C07281=1125.004,205.928,-65.608,-178.986,9.407,149.569
C07282=1125.008,205.679,-65.582,-178.988,9.404,149.569
C07283=1125.013,205.431,-65.557,-178.991,9.401,149.570
C07284=1125.017,205.181,-65.532,-178.994,9.398,149.570
C07285=1125.021,204.933,-65.506,-178.997,9.395,149.570
C07286=1125.026,204.684,-65.480,-179.000,9.392,149.570
C07287=1125.030,204.435,-65.456,-179.003,9.390,149.570
C07288=1125.035,204.187,-65.431,-179.006,9.387,149.570
C07289=1125.039,203.938,-65.405,-179.009,9.383,149.570
C07290=1125.044,203.690,-65.380,-179.012,9.380,149.570
C07291=1125.048,203.441,-65.354,-179.015,9.377,149.570
C07292=1125.053,203.192,-65.330,-179.018,9.375,149.570
C07293=1125.057,202.944,-65.305,-179.021,9.371,149.571
C07294=1125.062,202.694,-65.280,-179.024,9.368,149.571
C07295=1125.066,202.446,-65.254,-179.027,9.366,149.571
C07296=1125.070,202.197,-65.230,-179.031,9.362,149.571
C07297=1125.075,201.949,-65.204,-179.033,9.359,149.571
C07298=1125.080,201.699,-65.179,-179.037,9.356,149.571
C07299=1125.084,201.451,-65.154,-179.040,9.353,149.571
C07300=1125.088,201.202,-65.130,-179.043,9.349,149.571
C07301=1125.093,200.954,-65.104,-179.046,9.347,149.572
C07302=1125.097,200.705,-65.079,-179.050,9.343,149.572
C07303=1125.102,200.456,-65.055,-179.053,9.340,149.572
C07304=1125.106,200.208,-65.029,-179.056,9.337,149.572
C07305=1125.111,199.959,-65.005,-179.060,9.333,149.572
C07306=1125.116,199.710,-64.981,-179.063,9.331,149.572
C07307=1125.119,199.496,-64.959,-179.067,9.327,149.572
C07308=1125.124,199.282,-64.937,-179.069,9.324,149.572
C07309=1125.127,199.068,-64.916,-179.072,9.321,149.572
C07310=1125.131,198.854,-64.894,-179.075,9.318,149.573
C07311=1125.135,198.640,-64.873,-179.078,9.316,149.573
C07312=1125.139,198.426,-64.852,-179.081,9.313,149.573
C07313=1125.143,198.212,-64.831,-179.084,9.309,149.573
C07314=1125.146,197.998,-64.809,-179.087,9.306,149.573
C07315=1125.151,197.750,-64.785,-179.091,9.303,149.573
C07316=1125.155,197.501,-64.760,-179.094,9.299,149.573
C07317=1125.160,197.252,-64.735,-179.098,9.296,149.573
C07318=1125.164,197.003,-64.711,-179.101,9.292,149.573
C07319=1125.169,196.754,-64.686,-179.105,9.288,149.574
C07320=1125.173,196.506,-64.662,-179.109,9.284,149.574
C07321=1125.178,196.257,-64.637,-179.112,9.281,149.574
C07322=1125.182,196.008,-64.612,-179.114,9.278,149.574
C07323=1125.187,195.760,-64.588,-179.115,9.275,149.573
C07324=1125.191,195.511,-64.563,-179.117,9.273,149.573
C07325=1125.196,195.262,-64.539,-179.119,9.270,149.573
C07326=1125.201,195.013,-64.515,-179.121,9.268,149.573
C07327=1125.205,194.764,-64.490,-179.122,9.265,149.573
C07328=1125.210,194.516,-64.465,-179.124,9.263,149.573
C07329=1125.214,194.267,-64.441,-179.125,9.260,149.572
C07330=1125.218,194.018,-64.416,-179.127,9.258,149.572
C07331=1125.223,193.769,-64.392,-179.129,9.255,149.572
C07332=1125.228,193.521,-64.368,-179.131,9.253,149.572
C07333=1125.232,193.272,-64.343,-179.133,9.249,149.572
C07334=1125.237,193.023,-64.319,-179.135,9.247,149.572
C07335=1125.241,192.774,-64.294,-179.137,9.245,149.572
C07336=1125.246,192.526,-64.270,-179.138,9.242,149.572
C07337=1125.250,192.277,-64.245,-179.140,9.240,149.572
C07338=1125.255,192.028,-64.221,-179.142,9.236,149.572
C07339=1125.259,191.780,-64.197,-179.144,9.234,149.571
C07340=1125.264,191.531,-64.173,-179.146,9.231,149.571
C07341=1125.268,191.282,-64.148,-179.148,9.228,149.571
C07342=1125.273,191.033,-64.124,-179.150,9.226,149.571
C07343=1125.278,190.784,-64.100,-179.152,9.224,149.571
C07344=1125.282,190.535,-64.076,-179.155,9.221,149.571
C07345=1125.287,190.286,-64.051,-179.156,9.218,149.571
C07346=1125.291,190.038,-64.027,-179.159,9.215,149.571
C07347=1125.295,189.790,-64.003,-179.160,9.212,149.571
C07348=1125.300,189.540,-63.979,-179.163,9.209,149.571
C07349=1125.305,189.291,-63.954,-179.165,9.207,149.571
C07350=1125.309,189.043,-63.930,-179.167,9.204,149.571
C07351=1125.313,188.794,-63.906,-179.169,9.202,149.571
C07352=1125.319,188.546,-63.882,-179.172,9.198,149.571
C07353=1125.323,188.296,-63.858,-179.174,9.195,149.571
C07354=1125.327,188.047,-63.834,-179.176,9.193,149.570
C07355=1125.332,187.799,-63.810,-179.179,9.190,149.570
C07356=1125.337,187.550,-63.785,-179.181,9.188,149.570
C07357=1125.341,187.301,-63.762,-179.183,9.184,149.570
C07358=1125.346,187.053,-63.738,-179.186,9.181,149.570
C07359=1125.350,186.804,-63.713,-179.188,9.178,149.570
C07360=1125.355,186.554,-63.689,-179.190,9.176,149.570
C07361=1125.359,186.306,-63.665,-179.193,9.173,149.570
C07362=1125.364,186.057,-63.641,-179.196,9.170,149.570
C07363=1125.368,185.843,-63.620,-179.198,9.168,149.570
C07364=1125.372,185.629,-63.600,-179.200,9.165,149.570
C07365=1125.375,185.415,-63.580,-179.202,9.162,149.570
C07366=1125.379,185.200,-63.559,-179.204,9.160,149.570
C07367=1125.383,184.987,-63.538,-179.206,9.157,149.570
C07368=1125.387,184.772,-63.517,-179.208,9.155,149.570
C07369=1125.391,184.559,-63.497,-179.211,9.153,149.570
C07370=1125.395,184.344,-63.477,-179.213,9.149,149.570
C07371=1125.399,184.096,-63.452,-179.216,9.146,149.570
C07372=1125.404,183.847,-63.429,-179.218,9.143,149.570
C07373=1125.409,183.598,-63.405,-179.221,9.140,149.570
C07374=1125.413,183.349,-63.381,-179.224,9.137,149.570
C07375=1125.418,183.100,-63.357,-179.226,9.134,149.570
C07376=1125.423,182.851,-63.333,-179.229,9.131,149.570
C07377=1125.427,182.602,-63.309,-179.231,9.128,149.570
C07378=1125.432,182.353,-63.286,-179.235,9.125,149.570
C07379=1125.436,182.105,-63.262,-179.237,9.121,149.570
C07380=1125.441,181.856,-63.238,-179.240,9.118,149.570
C07381=1125.445,181.607,-63.215,-179.242,9.115,149.570
C07382=1125.450,181.359,-63.191,-179.246,9.112,149.570
C07383=1125.454,181.109,-63.168,-179.248,9.109,149.570
C07384=1125.459,180.861,-63.144,-179.251,9.105,149.570
C07385=1125.464,180.612,-63.120,-179.254,9.102,149.570
C07386=1125.468,180.363,-63.097,-179.257,9.099,149.570
C07387=1125.473,180.115,-63.073,-179.260,9.095,149.570
C07388=1125.477,179.866,-63.049,-179.263,9.092,149.570
C07389=1125.482,179.617,-63.026,-179.265,9.089,149.570
C07390=1125.486,179.368,-63.002,-179.269,9.085,149.570
C07391=1125.491,179.118,-62.978,-179.271,9.082,149.570
C07392=1125.495,178.869,-62.955,-179.274,9.079,149.570
C07393=1125.499,178.621,-62.932,-179.275,9.076,149.570
C07394=1125.504,178.372,-62.908,-179.278,9.073,149.570
C07395=1125.509,178.124,-62.885,-179.279,9.071,149.570
C07396=1125.514,177.875,-62.862,-179.282,9.067,149.570
C07397=1125.518,177.626,-62.838,-179.284,9.064,149.570
C07398=1125.523,177.377,-62.815,-179.286,9.062,149.569
C07399=1125.527,177.128,-62.791,-179.288,9.059,149.569
C07400=1125.532,176.879,-62.768,-179.291,9.055,149.569
C07401=1125.537,176.630,-62.744,-179.292,9.053,149.569
C07402=1125.541,176.382,-62.721,-179.295,9.050,149.569
C07403=1125.545,176.133,-62.698,-179.297,9.046,149.569
C07404=1125.550,175.884,-62.675,-179.299,9.044,149.569
C07405=1125.555,175.634,-62.651,-179.301,9.041,149.569
C07406=1125.559,175.386,-62.627,-179.304,9.037,149.569
C07407=1125.564,175.137,-62.604,-179.305,9.035,149.569
C07408=1125.568,174.888,-62.581,-179.308,9.032,149.569
C07409=1125.573,174.639,-62.558,-179.310,9.029,149.568
C07410=1125.577,174.390,-62.534,-179.312,9.026,149.568
C07411=1125.582,174.141,-62.511,-179.314,9.023,149.568
C07412=1125.586,173.893,-62.488,-179.317,9.020,149.568
C07413=1125.591,173.644,-62.465,-179.318,9.017,149.568
C07414=1125.596,173.395,-62.442,-179.321,9.014,149.568
C07415=1125.601,173.146,-62.419,-179.324,9.011,149.568
C07416=1125.605,172.897,-62.395,-179.326,9.008,149.568
C07417=1125.609,172.648,-62.372,-179.327,9.005,149.568
C07418=1125.614,172.399,-62.349,-179.330,9.002,149.568
C07419=1125.618,172.185,-62.330,-179.332,9.000,149.568
C07420=1125.622,171.971,-62.309,-179.334,8.996,149.567
C07421=1125.626,171.757,-62.289,-179.336,8.994,149.567
C07422=1125.631,171.542,-62.270,-179.338,8.991,149.567
C07423=1125.634,171.328,-62.250,-179.340,8.989,149.567
C07424=1125.638,171.114,-62.230,-179.342,8.986,149.567
C07425=1125.642,170.899,-62.210,-179.344,8.983,149.567
C07426=1125.646,170.685,-62.191,-179.346,8.981,149.567
C07427=1125.651,170.436,-62.167,-179.348,8.978,149.567
C07428=1125.655,170.188,-62.145,-179.351,8.975,149.567
C07429=1125.660,169.939,-62.122,-179.352,8.972,149.567
C07430=1125.665,169.690,-62.098,-179.355,8.969,149.567
C07431=1125.669,169.441,-62.076,-179.357,8.966,149.567
C07432=1125.674,169.192,-62.053,-179.359,8.962,149.566
C07433=1125.678,168.943,-62.029,-179.362,8.959,149.566
C07434=1125.683,168.695,-62.007,-179.364,8.956,149.566
C07435=1125.688,168.446,-61.984,-179.367,8.953,149.566
C07436=1125.692,168.196,-61.962,-179.368,8.950,149.566
C07437=1125.696,167.947,-61.938,-179.371,8.947,149.566
C07438=1125.702,167.699,-61.915,-179.373,8.944,149.566
C07439=1125.706,167.450,-61.893,-179.376,8.941,149.566
C07440=1125.711,167.201,-61.870,-179.378,8.937,149.566
C07441=1125.715,166.952,-61.847,-179.380,8.934,149.566
C07442=1125.719,166.703,-61.824,-179.383,8.931,149.566
C07443=1125.724,166.454,-61.802,-179.385,8.928,149.566
C07444=1125.729,166.205,-61.779,-179.388,8.925,149.565
C07445=1125.733,165.956,-61.757,-179.389,8.922,149.565
C07446=1125.739,165.708,-61.734,-179.392,8.919,149.565
C07447=1125.743,165.459,-61.711,-179.394,8.916,149.565
C07448=1125.748,165.209,-61.688,-179.397,8.913,149.565
C07449=1125.751,164.960,-61.665,-179.399,8.910,149.565
C07450=1125.757,164.711,-61.643,-179.402,8.906,149.565
C07451=1125.761,164.463,-61.620,-179.404,8.903,149.565
C07452=1125.766,164.214,-61.597,-179.406,8.900,149.565
C07453=1125.771,163.965,-61.575,-179.409,8.897,149.565
C07454=1125.775,163.716,-61.552,-179.411,8.893,149.564
C07455=1125.780,163.467,-61.530,-179.413,8.890,149.564
C07456=1125.784,163.218,-61.507,-179.416,8.887,149.564
C07457=1125.789,162.969,-61.485,-179.418,8.884,149.564
C07458=1125.793,162.720,-61.462,-179.420,8.880,149.564
C07459=1125.798,162.471,-61.440,-179.423,8.877,149.564
C07460=1125.803,162.223,-61.417,-179.426,8.874,149.564
C07461=1125.807,161.973,-61.395,-179.428,8.871,149.564
C07462=1125.812,161.724,-61.372,-179.430,8.868,149.564
C07463=1125.817,161.476,-61.350,-179.433,8.865,149.564
C07464=1125.822,161.226,-61.327,-179.435,8.860,149.563
C07465=1125.826,160.978,-61.305,-179.438,8.857,149.563
C07466=1125.830,160.729,-61.283,-179.440,8.854,149.563
C07467=1125.835,160.479,-61.260,-179.443,8.851,149.563
C07468=1125.840,160.231,-61.238,-179.445,8.847,149.563
C07469=1125.844,159.982,-61.216,-179.448,8.844,149.563
C07470=1125.849,159.733,-61.194,-179.450,8.841,149.563
C07471=1125.854,159.484,-61.171,-179.452,8.838,149.563
C07472=1125.858,159.235,-61.149,-179.455,8.834,149.563
C07473=1125.863,158.986,-61.127,-179.457,8.830,149.563
C07474=1125.868,158.736,-61.104,-179.460,8.827,149.562
C07475=1125.872,158.522,-61.085,-179.462,8.825,149.562
C07476=1125.876,158.308,-61.066,-179.464,8.821,149.562
C07477=1125.880,158.094,-61.047,-179.466,8.818,149.562
C07478=1125.884,157.879,-61.028,-179.468,8.816,149.562
C07479=1125.888,157.665,-61.009,-179.470,8.813,149.562
C07480=1125.892,157.450,-60.990,-179.472,8.810,149.562
C07481=1125.895,157.237,-60.971,-179.475,8.807,149.562
C07482=1125.899,157.022,-60.952,-179.477,8.804,149.562
C07483=1125.904,156.773,-60.929,-179.479,8.800,149.562
C07484=1125.909,156.524,-60.908,-179.482,8.797,149.561
C07485=1125.913,156.275,-60.886,-179.484,8.794,149.561
C07486=1125.918,156.026,-60.864,-179.487,8.790,149.561
C07487=1125.922,155.777,-60.841,-179.489,8.787,149.561
C07488=1125.928,155.528,-60.819,-179.492,8.783,149.561
C07489=1125.932,155.279,-60.797,-179.494,8.779,149.561
C07490=1125.937,155.030,-60.775,-179.497,8.776,149.561
C07491=1125.941,154.781,-60.753,-179.499,8.773,149.561
C07492=1125.946,154.532,-60.731,-179.502,8.769,149.561
C07493=1125.950,154.283,-60.709,-179.504,8.765,149.560
C07494=1125.955,154.034,-60.688,-179.507,8.762,149.560
C07495=1125.960,153.785,-60.666,-179.510,8.758,149.560
C07496=1125.964,153.537,-60.644,-179.512,8.755,149.560
C07497=1125.970,153.288,-60.622,-179.514,8.751,149.560
C07498=1125.974,153.038,-60.600,-179.517,8.747,149.560
C07499=1125.979,152.790,-60.578,-179.519,8.744,149.559
C07500=1125.983,152.540,-60.556,-179.522,8.741,149.559
C07501=1125.988,152.292,-60.534,-179.525,8.736,149.559
C07502=1125.993,152.042,-60.513,-179.527,8.733,149.559
C07503=1125.998,151.793,-60.491,-179.530,8.729,149.559
C07504=1126.003,151.544,-60.470,-179.532,8.726,149.559
C07505=1126.007,151.295,-60.447,-179.535,8.722,149.559
C07506=1126.012,151.046,-60.426,-179.537,8.718,149.558
C07507=1126.016,150.797,-60.404,-179.540,8.715,149.558
C07508=1126.021,150.548,-60.382,-179.542,8.711,149.558
C07509=1126.026,150.299,-60.361,-179.545,8.707,149.558
C07510=1126.030,150.050,-60.339,-179.548,8.703,149.558
C07511=1126.035,149.801,-60.317,-179.550,8.700,149.558
C07512=1126.040,149.553,-60.296,-179.552,8.696,149.557
C07513=1126.045,149.303,-60.274,-179.555,8.693,149.557
C07514=1126.049,149.054,-60.253,-179.558,8.688,149.557
C07515=1126.054,148.806,-60.232,-179.560,8.684,149.557
C07516=1126.058,148.556,-60.210,-179.563,8.681,149.557
C07517=1126.063,148.307,-60.189,-179.566,8.677,149.557
C07518=1126.068,148.058,-60.167,-179.568,8.673,149.556
C07519=1126.072,147.809,-60.145,-179.571,8.669,149.556
C07520=1126.077,147.560,-60.124,-179.573,8.666,149.556
C07521=1126.082,147.311,-60.102,-179.576,8.662,149.556
C07522=1126.086,147.061,-60.081,-179.578,8.657,149.556
C07523=1126.091,146.813,-60.060,-179.581,8.654,149.556
C07524=1126.096,146.564,-60.038,-179.584,8.650,149.555
C07525=1126.100,146.314,-60.017,-179.586,8.646,149.555
C07526=1126.105,146.066,-59.995,-179.588,8.642,149.555
C07527=1126.110,145.816,-59.974,-179.591,8.638,149.555
C07528=1126.115,145.568,-59.953,-179.594,8.634,149.555
C07529=1126.119,145.318,-59.932,-179.596,8.631,149.555
C07530=1126.124,145.069,-59.910,-179.599,8.626,149.554
C07531=1126.128,144.855,-59.892,-179.600,8.623,149.554
C07532=1126.132,144.640,-59.874,-179.602,8.620,149.554
C07533=1126.136,144.426,-59.855,-179.603,8.618,149.553
C07534=1126.140,144.212,-59.837,-179.604,8.615,149.553
C07535=1126.145,143.997,-59.819,-179.605,8.612,149.553
C07536=1126.148,143.783,-59.801,-179.606,8.609,149.552
C07537=1126.152,143.569,-59.782,-179.608,8.606,149.552
C07538=1126.156,143.354,-59.764,-179.609,8.603,149.552
C07539=1126.161,143.105,-59.743,-179.611,8.600,149.551
C07540=1126.166,142.855,-59.721,-179.612,8.597,149.551
C07541=1126.170,142.607,-59.701,-179.613,8.594,149.551
C07542=1126.175,142.358,-59.679,-179.615,8.590,149.550
C07543=1126.180,142.109,-59.658,-179.617,8.587,149.550
C07544=1126.185,141.860,-59.638,-179.618,8.583,149.550
C07545=1126.189,141.610,-59.616,-179.619,8.580,149.549
C07546=1126.194,141.361,-59.595,-179.621,8.577,149.549
C07547=1126.198,141.112,-59.575,-179.622,8.574,149.549
C07548=1126.203,140.864,-59.553,-179.624,8.570,149.548
C07549=1126.208,140.614,-59.532,-179.625,8.567,149.548
C07550=1126.213,140.365,-59.512,-179.627,8.564,149.548
C07551=1126.217,140.116,-59.489,-179.628,8.561,149.547
C07552=1126.222,139.867,-59.469,-179.631,8.557,149.547
C07553=1126.227,139.618,-59.448,-179.632,8.554,149.547
C07554=1126.232,139.368,-59.427,-179.634,8.550,149.546
C07555=1126.236,139.120,-59.406,-179.635,8.547,149.546
C07556=1126.241,138.871,-59.385,-179.637,8.544,149.546
C07557=1126.246,138.622,-59.365,-179.638,8.540,149.545
C07558=1126.250,138.372,-59.343,-179.640,8.537,149.545
C07559=1126.255,138.123,-59.322,-179.641,8.533,149.545
C07560=1126.260,137.874,-59.301,-179.643,8.531,149.544
C07561=1126.265,137.625,-59.280,-179.645,8.527,149.544
C07562=1126.269,137.376,-59.260,-179.646,8.524,149.544
C07563=1126.274,137.127,-59.239,-179.648,8.521,149.544
C07564=1126.279,136.878,-59.219,-179.649,8.518,149.543
C07565=1126.284,136.629,-59.197,-179.651,8.514,149.543
C07566=1126.288,136.380,-59.177,-179.652,8.511,149.542
C07567=1126.293,136.130,-59.155,-179.654,8.507,149.542
C07568=1126.297,135.881,-59.135,-179.656,8.505,149.542
C07569=1126.302,135.632,-59.114,-179.657,8.501,149.542
C07570=1126.307,135.383,-59.094,-179.659,8.497,149.541
C07571=1126.312,135.134,-59.073,-179.660,8.494,149.541
C07572=1126.316,134.885,-59.052,-179.662,8.491,149.541
C07573=1126.321,134.636,-59.031,-179.664,8.488,149.540
C07574=1126.326,134.387,-59.010,-179.665,8.484,149.540
C07575=1126.331,134.138,-58.989,-179.667,8.482,149.540
C07576=1126.335,133.889,-58.969,-179.669,8.478,149.540
C07577=1126.340,133.640,-58.948,-179.671,8.474,149.539
C07578=1126.345,133.391,-58.927,-179.672,8.471,149.539
C07579=1126.349,133.142,-58.907,-179.674,8.468,149.539
C07580=1126.354,132.893,-58.886,-179.675,8.465,149.538
C07581=1126.359,132.644,-58.866,-179.677,8.461,149.538
C07582=1126.364,132.395,-58.845,-179.679,8.458,149.538
C07583=1126.368,132.146,-58.824,-179.680,8.455,149.537
C07584=1126.373,131.896,-58.805,-179.682,8.451,149.537
C07585=1126.378,131.647,-58.784,-179.684,8.449,149.537
C07586=1126.383,131.398,-58.763,-179.685,8.445,149.536
C07587=1126.387,131.183,-58.746,-179.687,8.442,149.536
C07588=1126.391,130.969,-58.727,-179.688,8.439,149.536
C07589=1126.395,130.755,-58.710,-179.690,8.437,149.536
C07590=1126.399,130.540,-58.693,-179.691,8.434,149.536
C07591=1126.403,130.325,-58.674,-179.693,8.430,149.535
C07592=1126.407,130.110,-58.657,-179.695,8.428,149.535
C07593=1126.411,129.897,-58.639,-179.696,8.425,149.535
C07594=1126.415,129.681,-58.622,-179.697,8.422,149.534
C07595=1126.421,129.432,-58.601,-179.699,8.418,149.534
C07596=1126.425,129.183,-58.581,-179.701,8.416,149.534
C07597=1126.429,128.934,-58.561,-179.703,8.412,149.534
C07598=1126.434,128.685,-58.540,-179.704,8.409,149.533
C07599=1126.439,128.435,-58.520,-179.706,8.406,149.533
C07600=1126.444,128.187,-58.500,-179.708,8.402,149.533
C07601=1126.448,127.938,-58.479,-179.709,8.399,149.532
C07602=1126.453,127.688,-58.458,-179.711,8.395,149.532
C07603=1126.458,127.439,-58.439,-179.713,8.392,149.532
C07604=1126.463,127.191,-58.419,-179.714,8.389,149.532
C07605=1126.468,126.942,-58.398,-179.716,8.385,149.531
C07606=1126.473,126.692,-58.377,-179.718,8.382,149.531
C07607=1126.478,126.443,-58.358,-179.720,8.379,149.531
C07608=1126.482,126.194,-58.337,-179.722,8.376,149.531
C07609=1126.486,125.945,-58.317,-179.724,8.372,149.530
C07610=1126.491,125.695,-58.297,-179.725,8.368,149.530
C07611=1126.496,125.446,-58.276,-179.727,8.366,149.530
C07612=1126.501,125.197,-58.256,-179.729,8.362,149.530
C07613=1126.505,124.947,-58.236,-179.731,8.359,149.529
C07614=1126.511,124.699,-58.216,-179.732,8.355,149.529
C07615=1126.515,124.450,-58.196,-179.734,8.352,149.529
C07616=1126.520,124.201,-58.176,-179.736,8.348,149.528
C07617=1126.525,123.951,-58.155,-179.738,8.346,149.528
C07618=1126.530,123.702,-58.135,-179.740,8.342,149.528
C07619=1126.534,123.453,-58.115,-179.741,8.338,149.528
C07620=1126.538,123.204,-58.095,-179.743,8.335,149.527
C07621=1126.544,122.955,-58.075,-179.745,8.332,149.527
C07622=1126.548,122.706,-58.055,-179.747,8.329,149.527
C07623=1126.553,122.457,-58.035,-179.748,8.325,149.527
C07624=1126.557,122.208,-58.015,-179.751,8.321,149.526
C07625=1126.562,121.958,-57.995,-179.752,8.319,149.526
C07626=1126.567,121.709,-57.974,-179.754,8.315,149.526
C07627=1126.573,121.460,-57.955,-179.756,8.312,149.526
C07628=1126.577,121.211,-57.935,-179.758,8.308,149.525
C07629=1126.582,120.961,-57.915,-179.759,8.305,149.525
C07630=1126.586,120.713,-57.895,-179.761,8.302,149.525
C07631=1126.591,120.463,-57.875,-179.763,8.298,149.525
C07632=1126.596,120.215,-57.855,-179.765,8.295,149.524
C07633=1126.601,119.965,-57.835,-179.767,8.291,149.524
C07634=1126.606,119.716,-57.816,-179.768,8.288,149.524
C07635=1126.610,119.467,-57.795,-179.770,8.284,149.523
C07636=1126.615,119.218,-57.776,-179.773,8.281,149.523
C07637=1126.620,118.969,-57.756,-179.775,8.277,149.523
C07638=1126.625,118.719,-57.736,-179.776,8.274,149.523
C07639=1126.629,118.470,-57.716,-179.778,8.271,149.522
C07640=1126.634,118.221,-57.696,-179.780,8.267,149.522
C07641=1126.639,117.972,-57.677,-179.782,8.264,149.522
C07642=1126.644,117.722,-57.657,-179.784,8.260,149.522
C07643=1126.648,117.508,-57.640,-179.785,8.258,149.521
C07644=1126.652,117.293,-57.623,-179.787,8.255,149.521
C07645=1126.656,117.078,-57.606,-179.789,8.251,149.521
C07646=1126.661,116.864,-57.589,-179.790,8.249,149.521
C07647=1126.664,116.649,-57.572,-179.791,8.246,149.520
C07648=1126.668,116.435,-57.556,-179.793,8.242,149.520
C07649=1126.672,116.220,-57.538,-179.795,8.239,149.520
C07650=1126.677,116.006,-57.521,-179.796,8.237,149.520
C07651=1126.681,115.756,-57.502,-179.798,8.233,149.519
C07652=1126.686,115.507,-57.482,-179.800,8.230,149.519
C07653=1126.691,115.258,-57.463,-179.802,8.226,149.519
C07654=1126.696,115.009,-57.442,-179.804,8.223,149.519
C07655=1126.701,114.759,-57.423,-179.806,8.219,149.518
C07656=1126.705,114.511,-57.404,-179.808,8.215,149.518
C07657=1126.710,114.261,-57.384,-179.810,8.212,149.518
C07658=1126.715,114.011,-57.365,-179.812,8.208,149.518
C07659=1126.720,113.763,-57.345,-179.814,8.206,149.517
C07660=1126.724,113.514,-57.325,-179.815,8.202,149.517
C07661=1126.730,113.265,-57.306,-179.817,8.198,149.517
C07662=1126.734,113.016,-57.287,-179.819,8.195,149.517
C07663=1126.739,112.766,-57.267,-179.821,8.191,149.516
C07664=1126.744,112.517,-57.248,-179.823,8.187,149.516
C07665=1126.749,112.268,-57.228,-179.825,8.184,149.516
C07666=1126.753,112.018,-57.208,-179.827,8.180,149.516
C07667=1126.758,111.769,-57.190,-179.829,8.177,149.515
C07668=1126.763,111.520,-57.170,-179.831,8.173,149.515
C07669=1126.768,111.271,-57.151,-179.833,8.169,149.515
C07670=1126.773,111.021,-57.131,-179.835,8.166,149.514
C07671=1126.778,110.772,-57.111,-179.837,8.162,149.514
C07672=1126.782,110.523,-57.093,-179.840,8.158,149.514
C07673=1126.787,110.274,-57.073,-179.842,8.155,149.514
C07674=1126.792,110.025,-57.054,-179.844,8.150,149.514
C07675=1126.796,109.776,-57.035,-179.847,8.147,149.514
C07676=1126.802,109.527,-57.015,-179.850,8.143,149.513
C07677=1126.806,109.277,-56.996,-179.852,8.139,149.513
C07678=1126.810,109.028,-56.977,-179.854,8.135,149.513
C07679=1126.816,108.779,-56.957,-179.857,8.131,149.513
C07680=1126.821,108.529,-56.938,-179.859,8.127,149.512
C07681=1126.825,108.280,-56.920,-179.862,8.123,149.512
C07682=1126.830,108.031,-56.900,-179.864,8.120,149.512
C07683=1126.835,107.782,-56.881,-179.867,8.115,149.512
C07684=1126.839,107.533,-56.862,-179.869,8.112,149.512
C07685=1126.845,107.284,-56.842,-179.871,8.107,149.511
C07686=1126.849,107.034,-56.824,-179.873,8.104,149.511
C07687=1126.854,106.785,-56.805,-179.876,8.099,149.511
C07688=1126.859,106.535,-56.785,-179.878,8.096,149.510
C07689=1126.864,106.287,-56.766,-179.880,8.092,149.510
C07690=1126.869,106.037,-56.747,-179.882,8.088,149.510
C07691=1126.873,105.788,-56.729,-179.885,8.083,149.510
C07692=1126.878,105.539,-56.709,-179.887,8.080,149.509
C07693=1126.883,105.289,-56.691,-179.889,8.076,149.509
C07694=1126.888,105.040,-56.672,-179.891,8.072,149.509
C07695=1126.892,104.791,-56.653,-179.894,8.067,149.508
C07696=1126.898,104.542,-56.634,-179.896,8.064,149.508
C07697=1126.902,104.292,-56.615,-179.898,8.060,149.508
C07698=1126.907,104.044,-56.596,-179.901,8.056,149.508
C07699=1126.912,103.829,-56.580,-179.902,8.052,149.507
C07700=1126.916,103.614,-56.563,-179.904,8.050,149.507
C07701=1126.920,103.399,-56.547,-179.906,8.046,149.507
C07702=1126.924,103.185,-56.531,-179.908,8.043,149.507
C07703=1126.928,102.969,-56.514,-179.910,8.039,149.507
C07704=1126.932,102.755,-56.499,-179.911,8.035,149.506
C07705=1126.937,102.540,-56.482,-179.913,8.032,149.506
C07706=1126.941,102.326,-56.467,-179.915,8.029,149.506
C07707=1126.945,102.076,-56.448,-179.916,8.025,149.505
C07708=1126.951,101.827,-56.429,-179.919,8.021,149.505
C07709=1126.955,101.578,-56.410,-179.921,8.017,149.505
C07710=1126.960,101.328,-56.392,-179.923,8.013,149.504
C07711=1126.965,101.080,-56.373,-179.925,8.009,149.504
C07712=1126.969,100.830,-56.355,-179.927,8.005,149.504
C07713=1126.975,100.581,-56.335,-179.929,8.001,149.503
C07714=1126.979,100.332,-56.317,-179.931,7.997,149.503
C07715=1126.985,100.081,-56.298,-179.933,7.993,149.503
C07716=1126.989,99.833,-56.280,-179.935,7.990,149.502
C07717=1126.994,99.584,-56.262,-179.937,7.985,149.502
C07718=1126.999,99.334,-56.242,-179.939,7.981,149.502
C07719=1127.004,99.085,-56.224,-179.941,7.978,149.501
C07720=1127.009,98.836,-56.206,-179.942,7.974,149.501
C07721=1127.013,98.587,-56.187,-179.945,7.969,149.501
C07722=1127.018,98.337,-56.168,-179.947,7.966,149.500
C07723=1127.023,98.088,-56.150,-179.948,7.962,149.500
C07724=1127.028,97.839,-56.132,-179.950,7.958,149.499
C07725=1127.033,97.589,-56.113,-179.953,7.954,149.499
C07726=1127.038,97.340,-56.095,-179.954,7.950,149.499
C07727=1127.043,97.091,-56.077,-179.956,7.946,149.498
C07728=1127.047,96.842,-56.058,-179.957,7.942,149.498
C07729=1127.052,96.592,-56.039,-179.959,7.938,149.498
C07730=1127.057,96.343,-56.021,-179.962,7.934,149.497
C07731=1127.062,96.094,-56.003,-179.963,7.930,149.497
C07732=1127.067,95.845,-55.985,-179.965,7.926,149.496
C07733=1127.071,95.595,-55.966,-179.967,7.922,149.496
C07734=1127.077,95.346,-55.948,-179.968,7.918,149.496
C07735=1127.082,95.097,-55.930,-179.970,7.914,149.495
C07736=1127.087,94.847,-55.912,-179.972,7.911,149.495
C07737=1127.091,94.598,-55.893,-179.974,7.906,149.495
C07738=1127.095,94.349,-55.875,-179.976,7.902,149.494
C07739=1127.100,94.100,-55.857,-179.977,7.898,149.494
C07740=1127.106,93.850,-55.838,-179.979,7.894,149.493
C07741=1127.111,93.601,-55.820,-179.980,7.890,149.493
C07742=1127.115,93.351,-55.802,-179.982,7.887,149.492
C07743=1127.120,93.102,-55.784,-179.984,7.883,149.492
C07744=1127.125,92.853,-55.766,-179.985,7.879,149.492
C07745=1127.130,92.604,-55.748,-179.987,7.875,149.491
C07746=1127.135,92.355,-55.730,-179.988,7.871,149.491
C07747=1127.140,92.105,-55.712,-179.990,7.867,149.490
C07748=1127.144,91.856,-55.693,-179.992,7.863,149.490
C07749=1127.149,91.606,-55.675,-179.993,7.859,149.489
C07750=1127.155,91.357,-55.657,-179.995,7.855,149.489
C07751=1127.160,91.108,-55.639,-179.996,7.852,149.489
C07752=1127.164,90.859,-55.621,-179.998,7.848,149.488
C07753=1127.169,90.609,-55.603,-180.000,7.844,149.488
C07754=1127.174,90.360,-55.585,179.999,7.839,149.487
C07755=1127.178,90.145,-55.570,179.997,7.836,149.487
C07756=1127.182,89.930,-55.554,179.996,7.833,149.486
C07757=1127.186,89.715,-55.538,179.995,7.830,149.486
C07758=1127.190,89.501,-55.523,179.994,7.826,149.486
C07759=1127.194,89.286,-55.508,179.993,7.823,149.485
C07760=1127.199,89.071,-55.492,179.991,7.819,149.485
C07761=1127.203,88.856,-55.476,179.990,7.816,149.484
C07762=1127.207,88.641,-55.461,179.989,7.813,149.484
C07763=1127.212,88.392,-55.443,179.988,7.809,149.483
C07764=1127.217,88.143,-55.425,179.986,7.805,149.483
C07765=1127.222,87.893,-55.408,179.984,7.801,149.483
C07766=1127.227,87.644,-55.390,179.983,7.797,149.482
C07767=1127.232,87.395,-55.372,179.982,7.793,149.481
C07768=1127.237,87.146,-55.354,179.981,7.790,149.481
C07769=1127.242,86.896,-55.336,179.979,7.786,149.481
C07770=1127.246,86.646,-55.319,179.978,7.782,149.480
C07771=1127.251,86.397,-55.301,179.976,7.778,149.480
C07772=1127.256,86.148,-55.283,179.975,7.774,149.479
C07773=1127.261,85.899,-55.265,179.973,7.770,149.479
C07774=1127.266,85.649,-55.248,179.973,7.766,149.478
C07775=1127.271,85.400,-55.230,179.971,7.762,149.478
C07776=1127.276,85.151,-55.212,179.970,7.759,149.477
C07777=1127.281,84.901,-55.194,179.968,7.754,149.477
C07778=1127.286,84.652,-55.176,179.967,7.751,149.476
C07779=1127.290,84.403,-55.159,179.966,7.747,149.476
C07780=1127.295,84.154,-55.141,179.965,7.743,149.475
C07781=1127.300,83.904,-55.124,179.963,7.739,149.475
C07782=1127.305,83.655,-55.106,179.962,7.736,149.474
C07783=1127.310,83.405,-55.088,179.961,7.732,149.474
C07784=1127.315,83.156,-55.071,179.959,7.728,149.473
C07785=1127.319,82.907,-55.053,179.959,7.724,149.472
C07786=1127.324,82.658,-55.035,179.957,7.720,149.472
C07787=1127.330,82.408,-55.018,179.956,7.716,149.472
C07788=1127.334,82.159,-55.000,179.955,7.713,149.471
C07789=1127.340,81.909,-54.983,179.954,7.709,149.471
C07790=1127.344,81.660,-54.965,179.952,7.705,149.470
C07791=1127.349,81.411,-54.947,179.952,7.702,149.470
C07792=1127.355,81.162,-54.930,179.950,7.697,149.469
C07793=1127.360,80.913,-54.912,179.949,7.694,149.468
C07794=1127.364,80.663,-54.896,179.948,7.690,149.468
C07795=1127.369,80.414,-54.878,179.947,7.687,149.467
C07796=1127.374,80.164,-54.860,179.946,7.683,149.467
C07797=1127.379,79.915,-54.842,179.945,7.679,149.466
C07798=1127.384,79.665,-54.826,179.944,7.675,149.466
C07799=1127.388,79.416,-54.808,179.943,7.671,149.465
C07800=1127.394,79.166,-54.791,179.942,7.668,149.465
C07801=1127.399,78.917,-54.773,179.940,7.664,149.464
C07802=1127.403,78.668,-54.756,179.940,7.660,149.464
C07803=1127.408,78.419,-54.738,179.938,7.657,149.463
C07804=1127.413,78.169,-54.721,179.938,7.653,149.462
C07805=1127.418,77.921,-54.704,179.936,7.649,149.462
C07806=1127.423,77.671,-54.686,179.936,7.646,149.461
C07807=1127.428,77.422,-54.668,179.935,7.641,149.461
C07808=1127.433,77.172,-54.652,179.934,7.638,149.460
C07809=1127.438,76.922,-54.634,179.933,7.635,149.460
C07810=1127.443,76.673,-54.617,179.932,7.631,149.459
C07811=1127.447,76.458,-54.602,179.931,7.628,149.459
C07812=1127.451,76.243,-54.587,179.929,7.624,149.458
C07813=1127.455,76.028,-54.572,179.928,7.621,149.458
C07814=1127.460,75.814,-54.557,179.927,7.618,149.458
C07815=1127.464,75.599,-54.543,179.926,7.614,149.457
C07816=1127.468,75.384,-54.527,179.925,7.611,149.457
C07817=1127.473,75.169,-54.513,179.923,7.607,149.456
C07818=1127.476,74.954,-54.499,179.922,7.604,149.456
C07819=1127.481,74.704,-54.481,179.920,7.600,149.455
C07820=1127.486,74.455,-54.463,179.919,7.596,149.455
C07821=1127.492,74.206,-54.447,179.917,7.592,149.455
C07822=1127.496,73.957,-54.429,179.916,7.588,149.454
C07823=1127.501,73.707,-54.412,179.915,7.584,149.453
C07824=1127.506,73.457,-54.395,179.913,7.580,149.453
C07825=1127.511,73.208,-54.378,179.911,7.576,149.453
C07826=1127.516,72.959,-54.360,179.910,7.572,149.452
C07827=1127.521,72.710,-54.344,179.909,7.568,149.452
C07828=1127.526,72.460,-54.327,179.907,7.564,149.451
C07829=1127.530,72.211,-54.310,179.906,7.560,149.451
C07830=1127.536,71.961,-54.293,179.905,7.556,149.450
C07831=1127.540,71.713,-54.276,179.903,7.552,149.450
C07832=1127.546,71.463,-54.259,179.901,7.548,149.449
C07833=1127.550,71.213,-54.242,179.900,7.544,149.449
C07834=1127.555,70.964,-54.225,179.899,7.540,149.448
C07835=1127.560,70.714,-54.208,179.897,7.536,149.448
C07836=1127.566,70.465,-54.191,179.896,7.532,149.447
C07837=1127.570,70.216,-54.175,179.894,7.527,149.447
C07838=1127.575,69.966,-54.157,179.893,7.524,149.446
C07839=1127.580,69.718,-54.140,179.891,7.520,149.446
C07840=1127.585,69.468,-54.123,179.890,7.516,149.445
C07841=1127.590,69.218,-54.106,179.889,7.511,149.445
C07842=1127.594,68.969,-54.090,179.888,7.508,149.444
C07843=1127.600,68.720,-54.073,179.886,7.504,149.444
C07844=1127.605,68.470,-54.056,179.884,7.500,149.443
C07845=1127.610,68.221,-54.039,179.883,7.496,149.443
C07846=1127.615,67.972,-54.022,179.882,7.492,149.442
C07847=1127.619,67.722,-54.006,179.880,7.488,149.442
C07848=1127.625,67.472,-53.989,179.879,7.484,149.441
C07849=1127.629,67.223,-53.972,179.878,7.480,149.441
C07850=1127.634,66.974,-53.956,179.876,7.476,149.440
C07851=1127.639,66.724,-53.938,179.875,7.472,149.440
C07852=1127.644,66.475,-53.922,179.873,7.468,149.439
C07853=1127.649,66.226,-53.905,179.872,7.464,149.439
C07854=1127.654,65.976,-53.888,179.870,7.460,149.439
C07855=1127.659,65.727,-53.871,179.869,7.456,149.438
C07856=1127.664,65.477,-53.856,179.867,7.452,149.437
C07857=1127.669,65.228,-53.839,179.866,7.448,149.437
C07858=1127.674,64.978,-53.822,179.865,7.444,149.436
C07859=1127.679,64.729,-53.806,179.863,7.440,149.436
C07860=1127.684,64.480,-53.788,179.862,7.436,149.436
C07861=1127.689,64.231,-53.772,179.861,7.432,149.435
C07862=1127.693,63.981,-53.755,179.859,7.428,149.434
C07863=1127.698,63.731,-53.739,179.857,7.424,149.434
C07864=1127.704,63.482,-53.722,179.856,7.420,149.433
C07865=1127.709,63.233,-53.706,179.855,7.416,149.433
C07866=1127.713,62.983,-53.689,179.853,7.412,149.433
C07867=1127.718,62.769,-53.675,179.852,7.409,149.432
C07868=1127.722,62.553,-53.661,179.851,7.405,149.432
C07869=1127.726,62.338,-53.646,179.850,7.402,149.431
C07870=1127.731,62.124,-53.632,179.849,7.399,149.431
C07871=1127.735,61.908,-53.618,179.847,7.395,149.430
C07872=1127.739,61.693,-53.604,179.846,7.392,149.430
C07873=1127.744,61.478,-53.590,179.845,7.388,149.430
C07874=1127.748,61.263,-53.576,179.844,7.385,149.429
C07875=1127.752,61.014,-53.559,179.843,7.380,149.428
C07876=1127.757,60.765,-53.543,179.841,7.376,149.428
C07877=1127.763,60.514,-53.526,179.840,7.372,149.427
C07878=1127.768,60.266,-53.510,179.838,7.368,149.427
C07879=1127.772,60.016,-53.494,179.837,7.364,149.427
C07880=1127.778,59.767,-53.478,179.836,7.360,149.426
C07881=1127.782,59.517,-53.461,179.834,7.356,149.425
C07882=1127.788,59.268,-53.446,179.833,7.352,149.425
C07883=1127.792,59.018,-53.429,179.832,7.348,149.424
C07884=1127.797,58.770,-53.413,179.830,7.344,149.424
C07885=1127.803,58.519,-53.396,179.829,7.340,149.423
C07886=1127.808,58.270,-53.380,179.827,7.336,149.423
C07887=1127.813,58.020,-53.364,179.826,7.332,149.422
C07888=1127.818,57.772,-53.348,179.825,7.327,149.422
C07889=1127.822,57.522,-53.331,179.823,7.324,149.421
C07890=1127.827,57.273,-53.315,179.822,7.319,149.421
C07891=1127.832,57.023,-53.299,179.820,7.315,149.420
C07892=1127.837,56.774,-53.283,179.819,7.311,149.420
C07893=1127.842,56.524,-53.266,179.818,7.307,149.419
C07894=1127.847,56.275,-53.251,179.816,7.303,149.419
C07895=1127.852,56.025,-53.234,179.815,7.299,149.418
C07896=1127.857,55.776,-53.219,179.814,7.295,149.418
C07897=1127.862,55.526,-53.202,179.812,7.291,149.417
C07898=1127.867,55.277,-53.186,179.812,7.288,149.417
C07899=1127.871,55.028,-53.170,179.810,7.284,149.416
C07900=1127.877,54.778,-53.154,179.809,7.279,149.416
C07901=1127.882,54.529,-53.138,179.807,7.275,149.415
C07902=1127.887,54.279,-53.122,179.806,7.271,149.415
C07903=1127.892,54.030,-53.106,179.805,7.267,149.414
C07904=1127.897,53.780,-53.090,179.804,7.263,149.413
C07905=1127.902,53.531,-53.074,179.802,7.259,149.413
C07906=1127.907,53.282,-53.058,179.801,7.255,149.412
C07907=1127.912,53.032,-53.042,179.799,7.251,149.412
C07908=1127.917,52.783,-53.026,179.798,7.247,149.411
C07909=1127.922,52.533,-53.010,179.797,7.243,149.411
C07910=1127.927,52.284,-52.994,179.796,7.238,149.410
C07911=1127.932,52.034,-52.978,179.794,7.234,149.410
C07912=1127.937,51.784,-52.962,179.793,7.230,149.409
C07913=1127.942,51.536,-52.946,179.791,7.226,149.409
C07914=1127.947,51.286,-52.931,179.790,7.222,149.408
C07915=1127.952,51.036,-52.915,179.789,7.218,149.408
C07916=1127.957,50.787,-52.899,179.788,7.214,149.407
C07917=1127.962,50.537,-52.883,179.786,7.210,149.407
C07918=1127.967,50.288,-52.867,179.785,7.205,149.406
C07919=1127.972,50.039,-52.852,179.783,7.202,149.406
C07920=1127.976,49.789,-52.836,179.782,7.197,149.405
C07921=1127.982,49.540,-52.820,179.781,7.193,149.404
C07922=1127.987,49.291,-52.804,179.780,7.189,149.404
C07923=1127.991,49.075,-52.791,179.778,7.185,149.403
C07924=1127.995,48.861,-52.777,179.777,7.182,149.403
C07925=1128.000,48.645,-52.763,179.776,7.178,149.403
C07926=1128.005,48.430,-52.750,179.775,7.175,149.402
C07927=1128.008,48.215,-52.736,179.774,7.171,149.401
C07928=1128.013,48.000,-52.723,179.773,7.167,149.401
C07929=1128.017,47.784,-52.710,179.772,7.164,149.401
C07930=1128.021,47.570,-52.696,179.770,7.160,149.400
C07931=1128.027,47.320,-52.681,179.769,7.156,149.400
C07932=1128.031,47.070,-52.665,179.768,7.152,149.399
C07933=1128.037,46.821,-52.649,179.767,7.148,149.398
C07934=1128.041,46.572,-52.634,179.766,7.144,149.398
C07935=1128.046,46.322,-52.618,179.764,7.140,149.397
C07936=1128.052,46.072,-52.603,179.763,7.135,149.397
C07937=1128.057,45.823,-52.587,179.761,7.131,149.396
C07938=1128.062,45.574,-52.572,179.760,7.127,149.396
C07939=1128.066,45.324,-52.556,179.759,7.123,149.395
C07940=1128.072,45.074,-52.540,179.758,7.119,149.395
C07941=1128.076,44.825,-52.525,179.757,7.115,149.394
C07942=1128.082,44.576,-52.510,179.755,7.111,149.394
C07943=1128.087,44.326,-52.494,179.754,7.106,149.393
C07944=1128.091,44.077,-52.479,179.753,7.102,149.392
C07945=1128.097,43.827,-52.463,179.751,7.098,149.392
C07946=1128.102,43.578,-52.448,179.750,7.094,149.391
C07947=1128.107,43.329,-52.433,179.749,7.090,149.391
C07948=1128.111,43.079,-52.417,179.748,7.086,149.390
C07949=1128.117,42.829,-52.401,179.747,7.081,149.389
C07950=1128.121,42.580,-52.386,179.745,7.077,149.389
C07951=1128.127,42.331,-52.371,179.744,7.073,149.388
C07952=1128.131,42.082,-52.356,179.743,7.069,149.388
C07953=1128.136,41.831,-52.340,179.741,7.065,149.387
C07954=1128.142,41.581,-52.325,179.740,7.061,149.387
C07955=1128.147,41.332,-52.310,179.739,7.056,149.386
C07956=1128.152,41.083,-52.294,179.738,7.052,149.385
C07957=1128.157,40.834,-52.279,179.737,7.048,149.385
C07958=1128.162,40.584,-52.264,179.735,7.044,149.384
C07959=1128.167,40.335,-52.249,179.734,7.039,149.384
C07960=1128.172,40.085,-52.233,179.733,7.036,149.383
C07961=1128.177,39.835,-52.218,179.732,7.031,149.383
C07962=1128.182,39.586,-52.203,179.731,7.027,149.382
C07963=1128.187,39.337,-52.187,179.730,7.023,149.381
C07964=1128.192,39.087,-52.173,179.728,7.019,149.381
C07965=1128.198,38.838,-52.157,179.727,7.014,149.380
C07966=1128.202,38.589,-52.142,179.726,7.010,149.380
C07967=1128.208,38.339,-52.127,179.724,7.006,149.379
C07968=1128.213,38.089,-52.113,179.723,7.002,149.379
C07969=1128.217,37.839,-52.097,179.722,6.997,149.378
C07970=1128.222,37.590,-52.082,179.721,6.992,149.377
C07971=1128.228,37.340,-52.067,179.719,6.988,149.377
C07972=1128.232,37.091,-52.052,179.718,6.984,149.376
C07973=1128.238,36.842,-52.036,179.717,6.980,149.376
C07974=1128.243,36.592,-52.022,179.716,6.976,149.375
C07975=1128.247,36.343,-52.007,179.715,6.971,149.374
C07976=1128.253,36.094,-51.991,179.713,6.967,149.374
C07977=1128.258,35.844,-51.977,179.712,6.963,149.373
C07978=1128.263,35.594,-51.961,179.711,6.959,149.373
C07979=1128.268,35.379,-51.948,179.711,6.955,149.372
C07980=1128.271,35.164,-51.936,179.709,6.951,149.371
C07981=1128.276,34.949,-51.923,179.708,6.948,149.371
C07982=1128.280,34.734,-51.910,179.707,6.944,149.370
C07983=1128.284,34.518,-51.897,179.706,6.941,149.370
C07984=1128.289,34.303,-51.884,179.705,6.936,149.369
C07985=1128.294,34.088,-51.871,179.704,6.933,149.369
C07986=1128.298,33.873,-51.859,179.703,6.929,149.368
C07987=1128.303,33.623,-51.844,179.702,6.925,149.368
C07988=1128.308,33.374,-51.829,179.701,6.921,149.367
C07989=1128.313,33.125,-51.814,179.699,6.916,149.367
C07990=1128.318,32.875,-51.800,179.698,6.912,149.366
C07991=1128.323,32.625,-51.785,179.697,6.908,149.365
C07992=1128.328,32.376,-51.770,179.696,6.903,149.365
C07993=1128.333,32.126,-51.755,179.695,6.899,149.364
C07994=1128.338,31.877,-51.740,179.694,6.895,149.363
C07995=1128.343,31.628,-51.725,179.692,6.890,149.363
C07996=1128.349,31.378,-51.711,179.691,6.885,149.362
C07997=1128.354,31.128,-51.696,179.690,6.881,149.362
C07998=1128.358,30.879,-51.681,179.689,6.877,149.361
C07999=1128.363,30.629,-51.667,179.688,6.873,149.360
C08000=1128.369,30.380,-51.651,179.687,6.868,149.360
C08001=1128.374,30.130,-51.637,179.686,6.864,149.359
C08002=1128.379,29.880,-51.623,179.685,6.860,149.358
C08003=1128.383,29.631,-51.608,179.684,6.856,149.358
C08004=1128.389,29.381,-51.593,179.682,6.851,149.357
C08005=1128.394,29.131,-51.579,179.681,6.847,149.356
C08006=1128.399,28.882,-51.564,179.680,6.843,149.356
C08007=1128.404,28.633,-51.549,179.679,6.837,149.355
C08008=1128.408,28.383,-51.535,179.678,6.833,149.354
C08009=1128.414,28.134,-51.520,179.677,6.829,149.354
C08010=1128.419,27.884,-51.506,179.676,6.825,149.353
C08011=1128.424,27.635,-51.491,179.674,6.820,149.352
C08012=1128.429,27.385,-51.477,179.673,6.816,149.352
C08013=1128.434,27.136,-51.462,179.672,6.812,149.351
C08014=1128.439,26.886,-51.448,179.671,6.807,149.351
C08015=1128.445,26.636,-51.433,179.670,6.803,149.350
C08016=1128.450,26.386,-51.419,179.669,6.798,149.349
C08017=1128.455,26.137,-51.405,179.668,6.794,149.349
C08018=1128.460,25.888,-51.390,179.666,6.789,149.348
C08019=1128.465,25.639,-51.376,179.665,6.785,149.347
C08020=1128.470,25.389,-51.361,179.664,6.781,149.347
C08021=1128.475,25.139,-51.347,179.664,6.776,149.346
C08022=1128.480,24.890,-51.333,179.663,6.772,149.345
C08023=1128.486,24.640,-51.318,179.662,6.767,149.345
C08024=1128.491,24.391,-51.303,179.661,6.763,149.344
C08025=1128.495,24.141,-51.289,179.659,6.758,149.343
C08026=1128.500,23.892,-51.275,179.658,6.753,149.343
C08027=1128.505,23.642,-51.260,179.657,6.749,149.342
C08028=1128.510,23.392,-51.246,179.656,6.745,149.341
C08029=1128.516,23.143,-51.232,179.655,6.741,149.341
C08030=1128.521,22.894,-51.218,179.654,6.736,149.340
C08031=1128.526,22.644,-51.204,179.653,6.732,149.339
C08032=1128.531,22.394,-51.189,179.652,6.726,149.338
C08033=1128.536,22.144,-51.175,179.650,6.722,149.338
C08034=1128.541,21.895,-51.161,179.649,6.718,149.337
C08035=1128.546,21.680,-51.149,179.649,6.714,149.337
C08036=1128.549,21.464,-51.136,179.648,6.710,149.336
C08037=1128.554,21.249,-51.124,179.646,6.706,149.335
C08038=1128.559,21.034,-51.112,179.646,6.702,149.335
C08039=1128.563,20.819,-51.099,179.645,6.698,149.334
C08040=1128.567,20.603,-51.088,179.645,6.695,149.333
C08041=1128.571,20.388,-51.076,179.643,6.690,149.333
C08042=1128.576,20.173,-51.064,179.643,6.687,149.332
C08043=1128.581,19.923,-51.049,179.641,6.682,149.332
C08044=1128.586,19.673,-51.035,179.640,6.677,149.331
C08045=1128.592,19.424,-51.021,179.639,6.673,149.330
C08046=1128.597,19.174,-51.007,179.638,6.669,149.330
C08047=1128.602,18.925,-50.993,179.638,6.664,149.329
C08048=1128.607,18.676,-50.979,179.637,6.660,149.328
C08049=1128.612,18.426,-50.965,179.635,6.654,149.327
C08050=1128.617,18.177,-50.951,179.634,6.650,149.327
C08051=1128.622,17.927,-50.937,179.633,6.645,149.326
C08052=1128.627,17.677,-50.923,179.632,6.641,149.325
C08053=1128.632,17.428,-50.909,179.631,6.637,149.325
C08054=1128.637,17.178,-50.895,179.630,6.631,149.324
C08055=1128.643,16.929,-50.881,179.629,6.627,149.323
C08056=1128.648,16.678,-50.867,179.628,6.623,149.322
C08057=1128.652,16.429,-50.853,179.628,6.618,149.322
C08058=1128.658,16.180,-50.840,179.626,6.614,149.321
C08059=1128.663,15.930,-50.825,179.625,6.609,149.320
C08060=1128.668,15.680,-50.812,179.624,6.604,149.319
C08061=1128.674,15.431,-50.798,179.623,6.599,149.319
C08062=1128.678,15.182,-50.784,179.622,6.595,149.318
C08063=1128.683,14.933,-50.770,179.622,6.590,149.317
C08064=1128.689,14.682,-50.757,179.621,6.586,149.317
C08065=1128.694,14.433,-50.742,179.619,6.581,149.316
C08066=1128.699,14.184,-50.728,179.618,6.576,149.315
C08067=1128.704,13.934,-50.716,179.618,6.572,149.314
C08068=1128.709,13.684,-50.701,179.617,6.567,149.314
C08069=1128.714,13.435,-50.687,179.615,6.562,149.313
C08070=1128.719,13.185,-50.674,179.615,6.557,149.312
C08071=1128.724,12.936,-50.660,179.614,6.553,149.311
C08072=1128.729,12.686,-50.646,179.613,6.548,149.310
C08073=1128.735,12.436,-50.633,179.612,6.544,149.310
C08074=1128.740,12.187,-50.619,179.611,6.539,149.309
C08075=1128.745,11.937,-50.606,179.610,6.534,149.308
C08076=1128.750,11.688,-50.592,179.609,6.529,149.307
C08077=1128.755,11.438,-50.578,179.608,6.525,149.307
C08078=1128.760,11.189,-50.565,179.607,6.520,149.306
C08079=1128.765,10.939,-50.551,179.606,6.515,149.305
C08080=1128.771,10.689,-50.537,179.605,6.511,149.304
C08081=1128.775,10.440,-50.524,179.604,6.506,149.304
C08082=1128.781,10.190,-50.511,179.603,6.501,149.303
C08083=1128.786,9.941,-50.496,179.602,6.496,149.302
C08084=1128.791,9.691,-50.483,179.602,6.492,149.301
C08085=1128.796,9.442,-50.469,179.601,6.487,149.300
C08086=1128.801,9.191,-50.456,179.600,6.482,149.300
C08087=1128.806,8.943,-50.443,179.599,6.477,149.299
C08088=1128.811,8.692,-50.429,179.598,6.473,149.298
C08089=1128.817,8.443,-50.416,179.597,6.468,149.297
C08090=1128.822,8.193,-50.402,179.596,6.463,149.297
C08091=1128.826,7.979,-50.391,179.596,6.459,149.296
C08092=1128.831,7.763,-50.380,179.595,6.456,149.295
C08093=1128.836,7.547,-50.368,179.596,6.452,149.294
C08094=1128.840,7.332,-50.356,179.595,6.448,149.294
C08095=1128.844,7.117,-50.344,179.595,6.443,149.293
C08096=1128.849,6.901,-50.333,179.594,6.440,149.292
C08097=1128.853,6.685,-50.322,179.594,6.436,149.291
C08098=1128.857,6.470,-50.310,179.594,6.432,149.291
C08099=1128.863,6.221,-50.297,179.593,6.428,149.290
C08100=1128.867,5.971,-50.283,179.593,6.423,149.289
C08101=1128.873,5.722,-50.270,179.592,6.418,149.288
C08102=1128.877,5.472,-50.257,179.592,6.414,149.287
C08103=1128.883,5.223,-50.243,179.591,6.410,149.286
C08104=1128.888,4.973,-50.230,179.591,6.405,149.286
C08105=1128.893,4.723,-50.217,179.590,6.400,149.285
C08106=1128.898,4.474,-50.204,179.590,6.397,149.284
C08107=1128.903,4.224,-50.190,179.590,6.392,149.283
C08108=1128.908,3.975,-50.177,179.589,6.387,149.282
C08109=1128.914,3.724,-50.164,179.589,6.382,149.281
C08110=1128.919,3.476,-50.150,179.589,6.378,149.280
C08111=1128.924,3.226,-50.137,179.588,6.374,149.280
C08112=1128.929,2.976,-50.124,179.587,6.369,149.279
C08113=1128.935,2.726,-50.111,179.587,6.365,149.278
C08114=1128.939,2.476,-50.098,179.587,6.361,149.277
C08115=1128.945,2.227,-50.084,179.586,6.356,149.276
C08116=1128.950,1.978,-50.072,179.585,6.352,149.275
C08117=1128.955,1.728,-50.058,179.585,6.347,149.275
C08118=1128.960,1.478,-50.045,179.584,6.342,149.274
C08119=1128.965,1.228,-50.032,179.584,6.338,149.273
C08120=1128.970,0.979,-50.019,179.584,6.334,149.272
C08121=1128.976,0.730,-50.006,179.583,6.329,149.271
C08122=1128.981,0.480,-49.992,179.582,6.324,149.270
C08123=1128.986,0.230,-49.980,179.582,6.320,149.269
C08124=1128.991,-0.019,-49.967,179.582,6.316,149.269
C08125=1128.996,-0.269,-49.954,179.581,6.311,149.268
C08126=1129.001,-0.519,-49.941,179.580,6.307,149.267
C08127=1129.007,-0.768,-49.927,179.580,6.302,149.266
C08128=1129.012,-1.018,-49.914,179.579,6.297,149.265
C08129=1129.017,-1.267,-49.902,179.578,6.293,149.265
C08130=1129.023,-1.517,-49.888,179.578,6.289,149.264
C08131=1129.027,-1.767,-49.875,179.578,6.284,149.263
C08132=1129.032,-2.016,-49.863,179.577,6.280,149.262
C08133=1129.038,-2.266,-49.850,179.576,6.275,149.261
C08134=1129.043,-2.516,-49.837,179.576,6.271,149.260
C08135=1129.048,-2.765,-49.824,179.575,6.266,149.260
C08136=1129.054,-3.015,-49.811,179.575,6.261,149.259
C08137=1129.058,-3.265,-49.798,179.574,6.257,149.258
C08138=1129.063,-3.514,-49.785,179.574,6.253,149.257
C08139=1129.068,-3.763,-49.773,179.573,6.248,149.256
C08140=1129.074,-4.013,-49.759,179.572,6.244,149.256
C08141=1129.079,-4.263,-49.746,179.572,6.239,149.255
C08142=1129.084,-4.512,-49.734,179.571,6.234,149.254
C08143=1129.090,-4.762,-49.721,179.570,6.230,149.253
C08144=1129.094,-5.012,-49.708,179.570,6.225,149.252
C08145=1129.099,-5.261,-49.695,179.569,6.220,149.251
C08146=1129.104,-5.511,-49.683,179.568,6.216,149.251
C08147=1129.111,-5.827,-49.667,179.567,6.210,149.250
C08148=1129.118,-6.143,-49.650,179.567,6.204,149.249
C08149=1129.125,-6.458,-49.634,179.566,6.199,149.248
C08150=1129.131,-6.774,-49.618,179.565,6.193,149.247
C08151=1129.136,-7.023,-49.605,179.564,6.188,149.246
C08152=1129.141,-7.273,-49.593,179.564,6.185,149.245
C08153=1129.146,-7.523,-49.580,179.564,6.180,149.244
C08154=1129.152,-7.772,-49.567,179.563,6.175,149.243
C08155=1129.177,-9.038,-49.501,179.448,6.358,149.317
C08156=1129.187,-9.458,-49.479,179.444,6.356,149.318
C08157=1129.191,-9.708,-49.466,179.441,6.356,149.319
C08158=1129.197,-9.958,-49.454,179.439,6.355,149.319
C08159=1129.202,-10.207,-49.442,179.436,6.354,149.320
C08160=1129.207,-10.457,-49.429,179.434,6.353,149.320
C08161=1129.213,-10.706,-49.416,179.431,6.352,149.321
C08162=1129.218,-10.956,-49.404,179.429,6.352,149.321
C08163=1129.223,-11.206,-49.391,179.427,6.351,149.322
C08164=1129.228,-11.456,-49.379,179.424,6.350,149.322
C08165=1129.233,-11.705,-49.366,179.422,6.349,149.323
C08166=1129.238,-11.955,-49.354,179.419,6.348,149.323
C08167=1129.243,-12.204,-49.342,179.417,6.348,149.324
C08168=1129.249,-12.454,-49.329,179.415,6.347,149.325
C08169=1129.253,-12.704,-49.316,179.412,6.346,149.325
C08170=1129.258,-12.953,-49.304,179.410,6.344,149.325
C08171=1129.264,-13.203,-49.292,179.407,6.344,149.326
C08172=1129.269,-13.452,-49.279,179.405,6.343,149.327
C08173=1129.274,-13.702,-49.267,179.403,6.342,149.327
C08174=1129.279,-13.951,-49.254,179.400,6.342,149.328
C08175=1129.285,-14.201,-49.241,179.398,6.341,149.328
C08176=1129.290,-14.452,-49.229,179.395,6.340,149.329
C08177=1129.295,-14.701,-49.216,179.393,6.339,149.329
C08178=1129.301,-14.951,-49.204,179.390,6.339,149.330
C08179=1129.306,-15.200,-49.192,179.388,6.338,149.330
C08180=1129.311,-15.450,-49.179,179.386,6.337,149.331
C08181=1129.316,-15.699,-49.167,179.383,6.337,149.332
C08182=1129.321,-15.949,-49.155,179.380,6.335,149.332
C08183=1129.327,-16.199,-49.143,179.378,6.334,149.332
C08184=1129.332,-16.448,-49.130,179.376,6.333,149.333
C08185=1129.337,-16.698,-49.118,179.373,6.333,149.334
C08186=1129.342,-16.947,-49.106,179.371,6.332,149.334
C08187=1129.347,-17.197,-49.093,179.369,6.331,149.335
C08188=1129.352,-17.447,-49.082,179.366,6.331,149.335
C08189=1129.357,-17.696,-49.069,179.363,6.329,149.336
C08190=1129.362,-17.946,-49.057,179.361,6.329,149.336
C08191=1129.367,-18.195,-49.044,179.359,6.328,149.337
C08192=1129.373,-18.445,-49.033,179.356,6.327,149.337
C08193=1129.378,-18.695,-49.020,179.354,6.327,149.338
C08194=1129.383,-18.945,-49.008,179.352,6.326,149.338
C08195=1129.388,-19.194,-48.996,179.349,6.325,149.339
C08196=1129.394,-19.444,-48.984,179.347,6.324,149.339
C08197=1129.399,-19.694,-48.972,179.344,6.323,149.340
C08198=1129.404,-19.943,-48.959,179.342,6.322,149.340
C08199=1129.410,-20.193,-48.947,179.340,6.322,149.341
C08200=1129.415,-20.442,-48.935,179.337,6.321,149.342
C08201=1129.420,-20.692,-48.923,179.335,6.320,149.342
C08202=1129.425,-20.941,-48.911,179.333,6.320,149.343
C08203=1129.430,-21.191,-48.899,179.330,6.319,149.343
C08204=1129.436,-21.441,-48.887,179.328,6.318,149.344
C08205=1129.441,-21.691,-48.874,179.325,6.317,149.344
C08206=1129.446,-21.941,-48.863,179.323,6.316,149.345
C08207=1129.451,-22.190,-48.850,179.320,6.316,149.345
C08208=1129.457,-22.440,-48.838,179.318,6.315,149.346
C08209=1129.461,-22.689,-48.827,179.316,6.314,149.346
C08210=1129.467,-22.939,-48.814,179.313,6.314,149.347
C08211=1129.472,-23.189,-48.802,179.311,6.313,149.347
C08212=1129.477,-23.439,-48.790,179.309,6.312,149.348
C08213=1129.483,-23.688,-48.778,179.306,6.311,149.349
C08214=1129.488,-23.938,-48.766,179.304,6.310,149.349
C08215=1129.493,-24.187,-48.755,179.301,6.309,149.350
C08216=1129.498,-24.437,-48.743,179.299,6.309,149.350
C08217=1129.504,-24.707,-48.730,179.297,6.308,149.351
C08218=1129.509,-24.977,-48.717,179.294,6.307,149.351
C08219=1129.515,-25.248,-48.704,179.291,6.306,149.352
C08220=1129.521,-25.518,-48.691,179.289,6.305,149.352
C08221=1129.526,-25.767,-48.678,179.286,6.305,149.353
C08222=1129.531,-26.017,-48.667,179.284,6.304,149.354
C08223=1129.537,-26.267,-48.655,179.282,6.303,149.354
C08224=1129.542,-26.517,-48.643,179.280,6.303,149.355
C08225=1129.546,-26.766,-48.631,179.277,6.302,149.355
C08226=1129.552,-27.015,-48.619,179.275,6.302,149.356
C08227=1129.557,-27.265,-48.608,179.273,6.301,149.356
C08228=1129.563,-27.515,-48.596,179.270,6.299,149.357
C08229=1129.567,-27.765,-48.584,179.267,6.299,149.357
C08230=1129.572,-28.014,-48.572,179.265,6.298,149.358
C08231=1129.578,-28.264,-48.560,179.263,6.297,149.358
C08232=1129.583,-28.513,-48.549,179.261,6.296,149.359
C08233=1129.589,-28.763,-48.537,179.258,6.296,149.359
C08234=1129.594,-29.013,-48.525,179.256,6.295,149.360
C08235=1129.599,-29.263,-48.513,179.254,6.294,149.360
C08236=1129.604,-29.512,-48.501,179.251,6.294,149.361
C08237=1129.609,-29.762,-48.489,179.249,6.293,149.362
C08238=1129.615,-30.012,-48.478,179.247,6.293,149.362
C08239=1129.620,-30.261,-48.467,179.244,6.292,149.363
C08240=1129.625,-30.511,-48.455,179.242,6.291,149.363
C08241=1129.631,-30.761,-48.443,179.240,6.291,149.364
C08242=1129.636,-31.010,-48.432,179.237,6.290,149.364
C08243=1129.641,-31.260,-48.420,179.235,6.288,149.365
C08244=1129.646,-31.510,-48.408,179.232,6.288,149.365
C08245=1129.651,-31.760,-48.396,179.230,6.287,149.366
C08246=1129.657,-32.009,-48.385,179.228,6.286,149.366
C08247=1129.662,-32.258,-48.373,179.225,6.285,149.367
C08248=1129.667,-32.508,-48.361,179.223,6.285,149.367
C08249=1129.672,-32.758,-48.350,179.221,6.284,149.368
C08250=1129.677,-33.008,-48.338,179.218,6.284,149.368
C08251=1129.683,-33.257,-48.326,179.216,6.283,149.369
C08252=1129.688,-33.506,-48.315,179.213,6.282,149.370
C08253=1129.693,-33.756,-48.303,179.211,6.282,149.370
C08254=1129.698,-34.006,-48.292,179.209,6.281,149.371
C08255=1129.703,-34.256,-48.280,179.206,6.280,149.371
C08256=1129.709,-34.506,-48.268,179.204,6.280,149.372
C08257=1129.714,-34.755,-48.257,179.202,6.279,149.372
C08258=1129.720,-35.005,-48.246,179.200,6.278,149.373
C08259=1129.724,-35.255,-48.235,179.197,6.278,149.373
C08260=1129.730,-35.505,-48.223,179.195,6.277,149.374
C08261=1129.735,-35.754,-48.212,179.193,6.276,149.374
C08262=1129.741,-36.004,-48.200,179.191,6.275,149.375
C08263=1129.745,-36.253,-48.189,179.188,6.275,149.376
C08264=1129.751,-36.503,-48.177,179.186,6.274,149.376
C08265=1129.755,-36.753,-48.166,179.184,6.273,149.376
C08266=1129.761,-37.002,-48.154,179.181,6.273,149.377
C08267=1129.766,-37.252,-48.143,179.179,6.272,149.378
C08268=1129.772,-37.502,-48.131,179.177,6.271,149.378
C08269=1129.777,-37.752,-48.120,179.174,6.271,149.379
C08270=1129.783,-38.001,-48.109,179.172,6.270,149.379
C08271=1129.787,-38.251,-48.098,179.170,6.270,149.380
C08272=1129.793,-38.501,-48.086,179.167,6.269,149.380
C08273=1129.797,-38.750,-48.074,179.165,6.268,149.381
C08274=1129.803,-39.000,-48.063,179.163,6.267,149.381
C08275=1129.808,-39.249,-48.052,179.160,6.267,149.382
C08276=1129.814,-39.500,-48.040,179.158,6.266,149.382
C08277=1129.819,-39.749,-48.029,179.156,6.265,149.383
C08278=1129.825,-39.999,-48.018,179.154,6.265,149.383
C08279=1129.829,-40.248,-48.006,179.151,6.264,149.384
C08280=1129.835,-40.499,-47.995,179.149,6.263,149.384
C08281=1129.840,-40.748,-47.984,179.147,6.263,149.385
C08282=1129.845,-40.997,-47.973,179.145,6.262,149.385
C08283=1129.850,-41.247,-47.961,179.142,6.261,149.386
C08284=1129.856,-41.496,-47.950,179.140,6.261,149.387
C08285=1129.862,-41.747,-47.939,179.137,6.260,149.387
C08286=1129.866,-41.996,-47.928,179.135,6.259,149.388
C08287=1129.871,-42.245,-47.917,179.133,6.259,149.388
C08288=1129.877,-42.496,-47.906,179.130,6.258,149.389
C08289=1129.882,-42.746,-47.894,179.128,6.257,149.389
C08290=1129.888,-42.995,-47.883,179.126,6.256,149.390
C08291=1129.893,-43.244,-47.871,179.123,6.256,149.390
C08292=1129.898,-43.495,-47.861,179.121,6.255,149.391
C08293=1129.904,-43.744,-47.849,179.119,6.254,149.391
C08294=1129.908,-43.993,-47.838,179.117,6.254,149.392
C08295=1129.913,-44.244,-47.827,179.114,6.253,149.393
C08296=1129.919,-44.493,-47.816,179.112,6.253,149.393
C08297=1129.924,-44.743,-47.805,179.110,6.252,149.394
C08298=1129.929,-44.993,-47.794,179.108,6.251,149.394
C08299=1129.935,-45.242,-47.783,179.105,6.251,149.395
C08300=1129.940,-45.492,-47.771,179.103,6.250,149.395
C08301=1129.945,-45.742,-47.761,179.101,6.249,149.396
C08302=1129.951,-45.991,-47.749,179.098,6.248,149.396
C08303=1129.956,-46.241,-47.739,179.096,6.248,149.397
C08304=1129.961,-46.490,-47.728,179.093,6.247,149.397
C08305=1129.967,-46.740,-47.716,179.091,6.246,149.398
C08306=1129.972,-46.991,-47.705,179.089,6.246,149.398
C08307=1129.977,-47.239,-47.694,179.087,6.245,149.399
C08308=1129.982,-47.490,-47.684,179.084,6.244,149.399
C08309=1129.988,-47.739,-47.672,179.082,6.244,149.400
C08310=1129.993,-47.989,-47.662,179.080,6.243,149.400
C08311=1129.998,-48.239,-47.650,179.078,6.243,149.401
C08312=1130.003,-48.488,-47.640,179.076,6.243,149.402
C08313=1130.009,-48.738,-47.628,179.073,6.242,149.402
C08314=1130.014,-48.988,-47.618,179.071,6.241,149.403
C08315=1130.019,-49.237,-47.607,179.069,6.240,149.403
C08316=1130.024,-49.488,-47.596,179.067,6.239,149.403
C08317=1130.030,-49.737,-47.585,179.064,6.239,149.404
C08318=1130.035,-49.987,-47.574,179.062,6.238,149.405
C08319=1130.040,-50.236,-47.563,179.060,6.238,149.405
C08320=1130.045,-50.486,-47.553,179.058,6.237,149.406
C08321=1130.051,-50.757,-47.541,179.055,6.236,149.406
C08322=1130.057,-51.028,-47.528,179.053,6.236,149.407
C08323=1130.063,-51.299,-47.516,179.050,6.235,149.408
C08324=1130.068,-51.569,-47.506,179.048,6.235,149.408
C08325=1130.073,-51.819,-47.494,179.046,6.234,149.408
C08326=1130.079,-52.069,-47.484,179.043,6.233,149.409
C08327=1130.084,-52.318,-47.472,179.041,6.233,149.410
C08328=1130.089,-52.569,-47.462,179.039,6.232,149.410
C08329=1130.095,-52.818,-47.451,179.036,6.231,149.411
C08330=1130.099,-53.068,-47.440,179.034,6.230,149.411
C08331=1130.105,-53.317,-47.430,179.032,6.230,149.412
C08332=1130.110,-53.567,-47.418,179.029,6.229,149.412
C08333=1130.116,-53.817,-47.408,179.027,6.228,149.413
C08334=1130.121,-54.067,-47.397,179.026,6.228,149.413
C08335=1130.126,-54.316,-47.386,179.023,6.228,149.414
C08336=1130.131,-54.566,-47.376,179.021,6.227,149.414
C08337=1130.137,-54.816,-47.366,179.019,6.226,149.415
C08338=1130.142,-55.065,-47.354,179.016,6.226,149.415
C08339=1130.147,-55.315,-47.344,179.014,6.225,149.416
C08340=1130.152,-55.565,-47.333,179.012,6.224,149.416
C08341=1130.158,-55.814,-47.322,179.009,6.224,149.417
C08342=1130.163,-56.065,-47.311,179.007,6.223,149.418
C08343=1130.169,-56.314,-47.301,179.005,6.222,149.418
C08344=1130.174,-56.564,-47.290,179.003,6.222,149.419
C08345=1130.179,-56.813,-47.280,179.001,6.222,149.419
C08346=1130.184,-57.064,-47.269,178.998,6.221,149.420
C08347=1130.190,-57.313,-47.259,178.996,6.220,149.420
C08348=1130.195,-57.562,-47.248,178.994,6.220,149.421
C08349=1130.200,-57.812,-47.237,178.992,6.219,149.421
C08350=1130.206,-58.062,-47.227,178.989,6.219,149.422
C08351=1130.211,-58.312,-47.217,178.987,6.218,149.422
C08352=1130.216,-58.561,-47.206,178.985,6.217,149.423
C08353=1130.221,-58.811,-47.195,178.983,6.216,149.423
C08354=1130.227,-59.061,-47.185,178.981,6.216,149.424
C08355=1130.232,-59.311,-47.174,178.978,6.216,149.424
C08356=1130.237,-59.560,-47.163,178.976,6.215,149.425
C08357=1130.242,-59.809,-47.153,178.974,6.214,149.425
C08358=1130.247,-60.060,-47.143,178.972,6.214,149.426
C08359=1130.253,-60.309,-47.132,178.970,6.213,149.426
C08360=1130.258,-60.559,-47.122,178.967,6.212,149.427
C08361=1130.264,-60.809,-47.112,178.965,6.212,149.428
C08362=1130.268,-61.059,-47.100,178.963,6.212,149.428
C08363=1130.274,-61.308,-47.090,178.961,6.211,149.429
C08364=1130.279,-61.558,-47.080,178.959,6.210,149.429
C08365=1130.284,-61.808,-47.069,178.957,6.209,149.429
C08366=1130.290,-62.058,-47.059,178.954,6.209,149.430
C08367=1130.295,-62.308,-47.049,178.952,6.208,149.431
C08368=1130.301,-62.557,-47.038,178.950,6.207,149.431
C08369=1130.306,-62.806,-47.027,178.948,6.208,149.432
C08370=1130.311,-63.056,-47.017,178.946,6.207,149.432
C08371=1130.317,-63.306,-47.007,178.943,6.206,149.433
C08372=1130.322,-63.556,-46.996,178.941,6.206,149.433
C08373=1130.326,-63.806,-46.986,178.939,6.205,149.434
C08374=1130.332,-64.055,-46.976,178.936,6.204,149.434
C08375=1130.337,-64.305,-46.966,178.934,6.203,149.435
C08376=1130.343,-64.555,-46.955,178.932,6.204,149.435
C08377=1130.348,-64.804,-46.945,178.930,6.203,149.436
C08378=1130.353,-65.055,-46.935,178.928,6.202,149.436
C08379=1130.359,-65.304,-46.925,178.926,6.201,149.437
C08380=1130.364,-65.554,-46.914,178.923,6.201,149.437
C08381=1130.369,-65.804,-46.904,178.921,6.200,149.438
C08382=1130.375,-66.054,-46.894,178.919,6.200,149.439
C08383=1130.380,-66.303,-46.884,178.917,6.200,149.439
C08384=1130.385,-66.553,-46.873,178.915,6.199,149.440
C08385=1130.390,-66.803,-46.863,178.913,6.198,149.440
C08386=1130.396,-67.052,-46.853,178.910,6.197,149.441
C08387=1130.401,-67.302,-46.842,178.908,6.197,149.441
C08388=1130.407,-67.552,-46.832,178.906,6.197,149.442
C08389=1130.412,-67.801,-46.822,178.904,6.196,149.442
C08390=1130.417,-68.051,-46.812,178.902,6.195,149.443
C08391=1130.422,-68.301,-46.802,178.900,6.195,149.443
C08392=1130.428,-68.550,-46.792,178.897,6.194,149.444
C08393=1130.433,-68.800,-46.781,178.895,6.194,149.444
C08394=1130.438,-69.050,-46.771,178.893,6.194,149.445
C08395=1130.443,-69.299,-46.761,178.891,6.193,149.445
C08396=1130.449,-69.549,-46.751,178.889,6.192,149.446
C08397=1130.454,-69.799,-46.741,178.887,6.191,149.446
C08398=1130.460,-70.049,-46.731,178.884,6.191,149.447
C08399=1130.465,-70.299,-46.721,178.882,6.190,149.447
C08400=1130.470,-70.548,-46.711,178.880,6.190,149.448
C08401=1130.475,-70.798,-46.700,178.878,6.189,149.448
C08402=1130.481,-71.048,-46.690,178.876,6.189,149.449
C08403=1130.486,-71.297,-46.680,178.874,6.188,149.449
C08404=1130.492,-71.547,-46.670,178.871,6.187,149.450
C08405=1130.496,-71.798,-46.661,178.870,6.187,149.450
C08406=1130.502,-72.047,-46.650,178.867,6.187,149.451
C08407=1130.508,-72.297,-46.640,178.865,6.186,149.452
C08408=1130.513,-72.546,-46.630,178.863,6.185,149.452
C08409=1130.518,-72.796,-46.620,178.860,6.185,149.453
C08410=1130.523,-73.046,-46.610,178.859,6.185,149.453
C08411=1130.529,-73.296,-46.600,178.857,6.184,149.453
C08412=1130.535,-73.545,-46.590,178.854,6.183,149.454
C08413=1130.540,-73.795,-46.580,178.852,6.183,149.455
C08414=1130.545,-74.045,-46.570,178.850,6.182,149.455
C08415=1130.550,-74.294,-46.560,178.848,6.182,149.456
C08416=1130.555,-74.544,-46.551,178.846,6.181,149.456
C08417=1130.561,-74.794,-46.541,178.844,6.180,149.457
C08418=1130.566,-75.043,-46.530,178.841,6.180,149.457
C08419=1130.571,-75.294,-46.520,178.839,6.179,149.458
C08420=1130.577,-75.543,-46.511,178.837,6.179,149.458
C08421=1130.582,-75.793,-46.501,178.835,6.179,149.459
C08422=1130.588,-76.043,-46.490,178.833,6.178,149.459
C08423=1130.593,-76.292,-46.482,178.831,6.177,149.460
C08424=1130.598,-76.543,-46.471,178.829,6.177,149.460
C08425=1130.604,-76.813,-46.460,178.826,6.177,149.461
C08426=1130.610,-77.085,-46.450,178.824,6.176,149.461
C08427=1130.615,-77.357,-46.439,178.822,6.175,149.462
C08428=1130.622,-77.628,-46.428,178.819,6.175,149.463
C08429=1130.626,-77.878,-46.418,178.817,6.174,149.463
C08430=1130.632,-78.128,-46.409,178.815,6.173,149.464
C08431=1130.637,-78.378,-46.399,178.813,6.173,149.464
C08432=1130.643,-78.627,-46.389,178.811,6.173,149.465
C08433=1130.649,-78.877,-46.379,178.809,6.172,149.465
C08434=1130.653,-79.127,-46.370,178.807,6.171,149.465
C08435=1130.659,-79.376,-46.360,178.804,6.171,149.466
C08436=1130.664,-79.627,-46.350,178.802,6.171,149.467
C08437=1130.669,-79.876,-46.340,178.800,6.170,149.467
C08438=1130.675,-80.126,-46.331,178.798,6.169,149.468
C08439=1130.680,-80.376,-46.321,178.796,6.169,149.468
C08440=1130.686,-80.625,-46.311,178.794,6.169,149.469
C08441=1130.691,-80.875,-46.302,178.792,6.168,149.469
C08442=1130.696,-81.125,-46.292,178.790,6.167,149.470
C08443=1130.702,-81.375,-46.282,178.787,6.167,149.470
C08444=1130.706,-81.625,-46.272,178.786,6.167,149.471
C08445=1130.712,-81.874,-46.262,178.783,6.166,149.471
C08446=1130.717,-82.124,-46.253,178.781,6.165,149.472
C08447=1130.723,-82.374,-46.243,178.779,6.165,149.472
C08448=1130.728,-82.623,-46.234,178.777,6.165,149.473
C08449=1130.734,-82.873,-46.224,178.775,6.164,149.473
C08450=1130.739,-83.123,-46.215,178.773,6.163,149.474
C08451=1130.744,-83.372,-46.205,178.771,6.162,149.474
C08452=1130.750,-83.622,-46.196,178.769,6.163,149.475
C08453=1130.755,-83.872,-46.185,178.767,6.162,149.475
C08454=1130.760,-84.122,-46.176,178.764,6.161,149.476
C08455=1130.765,-84.372,-46.166,178.763,6.161,149.476
C08456=1130.770,-84.622,-46.157,178.761,6.161,149.477
C08457=1130.776,-84.871,-46.147,178.758,6.160,149.477
C08458=1130.781,-85.121,-46.138,178.756,6.159,149.478
C08459=1130.787,-85.371,-46.128,178.755,6.159,149.478
C08460=1130.792,-85.620,-46.119,178.752,6.158,149.479
C08461=1130.798,-85.870,-46.109,178.750,6.158,149.479
C08462=1130.803,-86.120,-46.100,178.748,6.157,149.480
C08463=1130.809,-86.370,-46.090,178.746,6.157,149.480
C08464=1130.814,-86.619,-46.081,178.744,6.156,149.481
C08465=1130.819,-86.869,-46.071,178.742,6.156,149.481
C08466=1130.824,-87.119,-46.062,178.740,6.156,149.482
C08467=1130.830,-87.369,-46.052,178.738,6.155,149.482
C08468=1130.834,-87.619,-46.042,178.736,6.154,149.483
C08469=1130.840,-87.869,-46.033,178.733,6.153,149.483
C08470=1130.846,-88.119,-46.024,178.732,6.154,149.484
C08471=1130.850,-88.368,-46.014,178.730,6.153,149.484
C08472=1130.856,-88.618,-46.005,178.727,6.152,149.485
C08473=1130.861,-88.868,-45.996,178.725,6.152,149.485
C08474=1130.866,-89.117,-45.986,178.723,6.152,149.486
C08475=1130.872,-89.367,-45.977,178.721,6.151,149.486
C08476=1130.877,-89.617,-45.967,178.719,6.150,149.487
C08477=1130.883,-89.867,-45.958,178.717,6.150,149.487
C08478=1130.888,-90.117,-45.949,178.715,6.149,149.488
C08479=1130.893,-90.366,-45.939,178.713,6.149,149.488
C08480=1130.899,-90.616,-45.930,178.711,6.149,149.489
C08481=1130.904,-90.866,-45.921,178.709,6.148,149.489
C08482=1130.910,-91.115,-45.910,178.707,6.147,149.490
C08483=1130.915,-91.365,-45.902,178.705,6.147,149.490
C08484=1130.920,-91.615,-45.893,178.702,6.147,149.491
C08485=1130.926,-91.865,-45.883,178.700,6.146,149.492
C08486=1130.931,-92.115,-45.874,178.698,6.145,149.492
C08487=1130.936,-92.364,-45.865,178.696,6.146,149.493
C08488=1130.942,-92.615,-45.855,178.694,6.145,149.493
C08489=1130.947,-92.864,-45.846,178.692,6.144,149.493
C08490=1130.952,-93.113,-45.837,178.691,6.144,149.494
C08491=1130.958,-93.363,-45.828,178.688,6.143,149.494
C08492=1130.964,-93.613,-45.819,178.686,6.143,149.495
C08493=1130.969,-93.863,-45.810,178.685,6.143,149.495
C08494=1130.974,-94.112,-45.800,178.682,6.142,149.496
C08495=1130.979,-94.362,-45.791,178.680,6.141,149.496
C08496=1130.985,-94.612,-45.782,178.679,6.141,149.497
C08497=1130.990,-94.862,-45.773,178.676,6.140,149.497
C08498=1130.995,-95.111,-45.763,178.674,6.140,149.498
C08499=1131.001,-95.361,-45.754,178.672,6.140,149.499
C08500=1131.006,-95.611,-45.745,178.670,6.139,149.499
C08501=1131.012,-95.861,-45.735,178.668,6.139,149.500
C08502=1131.017,-96.111,-45.726,178.665,6.138,149.500
C08503=1131.022,-96.361,-45.718,178.664,6.138,149.501
C08504=1131.027,-96.610,-45.708,178.662,6.137,149.501
C08505=1131.033,-96.860,-45.698,178.659,6.136,149.501
C08506=1131.039,-97.110,-45.690,178.658,6.136,149.502
C08507=1131.044,-97.359,-45.681,178.656,6.136,149.502
C08508=1131.049,-97.609,-45.672,178.653,6.135,149.503
C08509=1131.055,-97.859,-45.663,178.652,6.135,149.503
C08510=1131.060,-98.109,-45.654,178.650,6.134,149.504
C08511=1131.065,-98.359,-45.644,178.647,6.133,149.504
C08512=1131.070,-98.608,-45.635,178.646,6.133,149.505
C08513=1131.076,-98.859,-45.626,178.644,6.133,149.505
C08514=1131.081,-99.108,-45.617,178.642,6.133,149.506
C08515=1131.087,-99.358,-45.608,178.640,6.132,149.506
C08516=1131.092,-99.607,-45.599,178.638,6.131,149.507
C08517=1131.098,-99.858,-45.590,178.636,6.131,149.507
C08518=1131.103,-100.107,-45.581,178.633,6.131,149.508
C08519=1131.108,-100.357,-45.572,178.631,6.130,149.509
C08520=1131.113,-100.607,-45.563,178.630,6.130,149.509
C08521=1131.119,-100.857,-45.554,178.627,6.130,149.509
C08522=1131.124,-101.106,-45.546,178.625,6.129,149.510
C08523=1131.130,-101.356,-45.536,178.624,6.129,149.510
C08524=1131.135,-101.606,-45.527,178.621,6.128,149.511
C08525=1131.141,-101.856,-45.518,178.619,6.127,149.511
C08526=1131.146,-102.106,-45.510,178.618,6.127,149.512
C08527=1131.151,-102.356,-45.501,178.615,6.127,149.512
C08528=1131.156,-102.606,-45.492,178.613,6.126,149.513
C08529=1131.162,-102.877,-45.482,178.612,6.126,149.513
C08530=1131.169,-103.150,-45.472,178.609,6.125,149.514
C08531=1131.174,-103.422,-45.462,178.607,6.124,149.514
C08532=1131.180,-103.694,-45.452,178.605,6.124,149.515
C08533=1131.185,-103.944,-45.443,178.603,6.124,149.516
C08534=1131.190,-104.194,-45.434,178.601,6.123,149.516
C08535=1131.196,-104.444,-45.426,178.599,6.123,149.517
C08536=1131.202,-104.693,-45.418,178.597,6.123,149.517
C08537=1131.207,-104.943,-45.409,178.595,6.122,149.518
C08538=1131.212,-105.193,-45.400,178.593,6.122,149.518
C08539=1131.217,-105.443,-45.391,178.591,6.121,149.518
C08540=1131.222,-105.693,-45.382,178.589,6.121,149.519
C08541=1131.229,-105.942,-45.373,178.587,6.121,149.519
C08542=1131.234,-106.192,-45.364,178.585,6.120,149.520
C08543=1131.239,-106.442,-45.355,178.583,6.119,149.520
C08544=1131.244,-106.692,-45.346,178.581,6.119,149.521
C08545=1131.249,-106.942,-45.337,178.579,6.118,149.521
C08546=1131.255,-107.191,-45.329,178.577,6.118,149.522
C08547=1131.261,-107.441,-45.321,178.575,6.118,149.522
C08548=1131.266,-107.691,-45.312,178.573,6.117,149.523
C08549=1131.271,-107.941,-45.303,178.571,6.117,149.523
C08550=1131.277,-108.190,-45.294,178.569,6.116,149.524
C08551=1131.282,-108.440,-45.285,178.568,6.116,149.524
C08552=1131.287,-108.690,-45.276,178.565,6.116,149.525
C08553=1131.292,-108.940,-45.268,178.563,6.115,149.525
C08554=1131.298,-109.189,-45.260,178.562,6.115,149.526
C08555=1131.303,-109.439,-45.251,178.559,6.114,149.526
C08556=1131.309,-109.689,-45.242,178.558,6.114,149.527
C08557=1131.314,-109.939,-45.233,178.556,6.113,149.527
C08558=1131.320,-110.188,-45.224,178.553,6.113,149.528
C08559=1131.325,-110.438,-45.216,178.552,6.113,149.528
C08560=1131.330,-110.688,-45.207,178.550,6.112,149.529
C08561=1131.335,-110.938,-45.199,178.548,6.112,149.529
C08562=1131.341,-111.187,-45.190,178.546,6.111,149.530
C08563=1131.346,-111.437,-45.181,178.544,6.111,149.530
C08564=1131.352,-111.688,-45.173,178.542,6.111,149.531
C08565=1131.357,-111.938,-45.164,178.540,6.110,149.531
C08566=1131.363,-112.187,-45.155,178.538,6.110,149.532
C08567=1131.368,-112.437,-45.147,178.537,6.109,149.532
C08568=1131.373,-112.687,-45.138,178.534,6.108,149.532
C08569=1131.379,-112.936,-45.130,178.533,6.108,149.533
C08570=1131.384,-113.186,-45.121,178.531,6.107,149.533
C08571=1131.389,-113.436,-45.112,178.529,6.107,149.534
C08572=1131.395,-113.686,-45.104,178.527,6.107,149.534
C08573=1131.401,-113.936,-45.095,178.525,6.107,149.535
C08574=1131.406,-114.185,-45.086,178.523,6.106,149.535
C08575=1131.411,-114.436,-45.078,178.521,6.105,149.536
C08576=1131.417,-114.685,-45.070,178.519,6.105,149.536
C08577=1131.422,-114.935,-45.061,178.517,6.104,149.537
C08578=1131.427,-115.185,-45.052,178.515,6.104,149.537
C08579=1131.433,-115.434,-45.045,178.513,6.104,149.538
C08580=1131.438,-115.684,-45.036,178.512,6.104,149.538
C08581=1131.443,-115.934,-45.027,178.509,6.103,149.539
C08582=1131.449,-116.184,-45.019,178.507,6.102,149.539
C08583=1131.454,-116.434,-45.010,178.506,6.102,149.540
C08584=1131.459,-116.683,-45.001,178.503,6.102,149.540
C08585=1131.466,-116.933,-44.993,178.502,6.102,149.541
C08586=1131.471,-117.183,-44.985,178.500,6.101,149.541
C08587=1131.477,-117.433,-44.977,178.498,6.101,149.542
C08588=1131.481,-117.682,-44.968,178.496,6.100,149.542
C08589=1131.486,-117.932,-44.960,178.494,6.100,149.543
C08590=1131.492,-118.182,-44.952,178.493,6.099,149.543
C08591=1131.498,-118.432,-44.943,178.490,6.098,149.543
C08592=1131.503,-118.682,-44.935,178.489,6.098,149.544
C08593=1131.509,-118.931,-44.926,178.487,6.098,149.544
C08594=1131.514,-119.181,-44.917,178.485,6.098,149.545
C08595=1131.519,-119.431,-44.910,178.483,6.097,149.545
C08596=1131.525,-119.681,-44.901,178.481,6.097,149.546
C08597=1131.530,-119.931,-44.893,178.479,6.096,149.546
C08598=1131.536,-120.180,-44.884,178.477,6.096,149.547
C08599=1131.541,-120.431,-44.876,178.475,6.096,149.547
C08600=1131.546,-120.681,-44.867,178.473,6.095,149.548
C08601=1131.551,-120.929,-44.859,178.471,6.095,149.548
C08602=1131.557,-121.180,-44.851,178.469,6.094,149.549
C08603=1131.562,-121.430,-44.842,178.468,6.094,149.549
C08604=1131.568,-121.679,-44.834,178.465,6.094,149.550
C08605=1131.573,-121.929,-44.826,178.464,6.093,149.550
C08606=1131.579,-122.179,-44.818,178.462,6.092,149.550
C08607=1131.584,-122.429,-44.809,178.460,6.092,149.551
C08608=1131.589,-122.679,-44.801,178.458,6.092,149.551
C08609=1131.595,-122.928,-44.793,178.456,6.091,149.552
C08610=1131.600,-123.178,-44.785,178.454,6.091,149.552
C08611=1131.606,-123.428,-44.777,178.452,6.090,149.553
C08612=1131.611,-123.678,-44.768,178.451,6.090,149.553
C08613=1131.617,-123.927,-44.760,178.448,6.090,149.554
C08614=1131.622,-124.177,-44.752,178.447,6.090,149.554
C08615=1131.627,-124.428,-44.744,178.445,6.089,149.555
C08616=1131.633,-124.677,-44.736,178.444,6.089,149.555
C08617=1131.638,-124.927,-44.727,178.441,6.088,149.556
C08618=1131.643,-125.176,-44.720,178.440,6.088,149.556
C08619=1131.649,-125.427,-44.711,178.438,6.087,149.557
C08620=1131.654,-125.676,-44.703,178.436,6.087,149.557
C08621=1131.660,-125.926,-44.695,178.434,6.086,149.558
C08622=1131.665,-126.176,-44.687,178.432,6.087,149.558
C08623=1131.670,-126.426,-44.678,178.430,6.086,149.559
C08624=1131.676,-126.676,-44.670,178.428,6.086,149.559
C08625=1131.681,-126.925,-44.662,178.426,6.085,149.559
C08626=1131.686,-127.175,-44.654,178.425,6.085,149.560
C08627=1131.693,-127.425,-44.646,178.423,6.084,149.560
C08628=1131.698,-127.675,-44.637,178.421,6.084,149.561
C08629=1131.703,-127.925,-44.630,178.419,6.083,149.561
C08630=1131.708,-128.174,-44.621,178.417,6.083,149.562
C08631=1131.714,-128.424,-44.614,178.415,6.083,149.562
C08632=1131.719,-128.674,-44.606,178.413,6.082,149.563
C08633=1131.298,-128.685,-44.650,178.410,6.086,149.564
C08634=1131.293,-128.435,-44.658,178.413,6.086,149.564
C08635=1131.287,-128.186,-44.666,178.414,6.087,149.564
C08636=1131.282,-127.936,-44.674,178.416,6.087,149.563
C08637=1131.277,-127.686,-44.682,178.417,6.087,149.563
C08638=1131.271,-127.436,-44.691,178.420,6.088,149.562
C08639=1131.266,-127.186,-44.699,178.421,6.088,149.562
C08640=1131.261,-126.937,-44.707,178.423,6.089,149.561
C08641=1131.255,-126.687,-44.715,178.425,6.089,149.561
C08642=1131.249,-126.437,-44.723,178.427,6.089,149.560
C08643=1131.244,-126.187,-44.732,178.429,6.089,149.560
C08644=1131.239,-125.937,-44.739,178.431,6.091,149.559
C08645=1131.234,-125.688,-44.748,178.432,6.090,149.559
C08646=1131.228,-125.438,-44.755,178.434,6.091,149.558
C08647=1131.223,-125.188,-44.763,178.436,6.091,149.558
C08648=1131.217,-124.939,-44.772,178.438,6.092,149.557
C08649=1131.212,-124.688,-44.780,178.440,6.092,149.557
C08650=1131.207,-124.438,-44.789,178.442,6.093,149.556
C08651=1131.201,-124.189,-44.796,178.444,6.093,149.556
C08652=1131.196,-123.939,-44.805,178.446,6.093,149.555
C08653=1131.190,-123.689,-44.813,178.447,6.094,149.555
C08654=1131.185,-123.439,-44.821,178.449,6.094,149.555
C08655=1131.179,-123.190,-44.829,178.451,6.095,149.554
C08656=1131.174,-122.940,-44.838,178.453,6.095,149.554
C08657=1131.169,-122.689,-44.846,178.455,6.096,149.553
C08658=1131.163,-122.440,-44.854,178.457,6.096,149.553
C08659=1131.158,-122.190,-44.862,178.459,6.096,149.552
C08660=1131.153,-121.941,-44.870,178.460,6.096,149.552
C08661=1131.147,-121.691,-44.879,178.463,6.097,149.551
C08662=1131.142,-121.441,-44.888,178.464,6.097,149.551
C08663=1131.136,-121.191,-44.895,178.466,6.098,149.550
C08664=1131.131,-120.941,-44.904,178.468,6.098,149.550
C08665=1131.125,-120.692,-44.911,178.470,6.099,149.550
C08666=1131.120,-120.442,-44.920,178.471,6.099,149.549
C08667=1131.115,-120.191,-44.929,178.474,6.100,149.549
C08668=1131.109,-119.942,-44.937,178.476,6.100,149.548
C08669=1131.103,-119.692,-44.945,178.477,6.100,149.548
C08670=1131.098,-119.443,-44.953,178.480,6.101,149.547
C08671=1131.093,-119.193,-44.962,178.481,6.101,149.547
C08672=1131.088,-118.943,-44.970,178.483,6.102,149.546
C08673=1131.082,-118.693,-44.979,178.485,6.102,149.546
C08674=1131.077,-118.443,-44.987,178.487,6.102,149.545
C08675=1131.071,-118.193,-44.996,178.489,6.102,149.545
C08676=1131.066,-117.944,-45.003,178.491,6.103,149.544
C08677=1131.061,-117.694,-45.012,178.493,6.104,149.544
C08678=1131.056,-117.444,-45.021,178.495,6.104,149.543
C08679=1131.050,-117.194,-45.029,178.496,6.105,149.543
C08680=1131.044,-116.944,-45.038,178.498,6.105,149.542
C08681=1131.039,-116.695,-45.046,178.500,6.106,149.542
C08682=1131.033,-116.445,-45.054,178.502,6.106,149.541
C08683=1131.028,-116.195,-45.063,178.504,6.106,149.541
C08684=1131.022,-115.946,-45.072,178.506,6.107,149.540
C08685=1131.018,-115.696,-45.079,178.508,6.107,149.540
C08686=1131.012,-115.446,-45.088,178.510,6.108,149.540
C08687=1131.007,-115.197,-45.097,178.512,6.108,149.539
C08688=1131.001,-114.946,-45.105,178.514,6.109,149.539
C08689=1130.996,-114.696,-45.114,178.515,6.108,149.538
C08690=1130.990,-114.447,-45.122,178.518,6.109,149.538
C08691=1130.985,-114.197,-45.131,178.520,6.110,149.537
C08692=1130.980,-113.947,-45.139,178.521,6.110,149.537
C08693=1130.974,-113.698,-45.148,178.524,6.111,149.536
C08694=1130.968,-113.447,-45.156,178.525,6.111,149.536
C08695=1130.963,-113.197,-45.165,178.527,6.111,149.535
C08696=1130.958,-112.947,-45.174,178.529,6.111,149.535
C08697=1130.952,-112.698,-45.183,178.531,6.112,149.534
C08698=1130.947,-112.448,-45.191,178.533,6.113,149.534
C08699=1130.942,-112.198,-45.200,178.535,6.113,149.533
C08700=1130.936,-111.949,-45.208,178.537,6.113,149.533
C08701=1130.931,-111.699,-45.216,178.539,6.113,149.532
C08702=1130.926,-111.449,-45.225,178.540,6.115,149.532
C08703=1130.921,-111.199,-45.234,178.543,6.115,149.531
C08704=1130.915,-110.950,-45.242,178.544,6.115,149.531
C08705=1130.910,-110.700,-45.251,178.546,6.116,149.530
C08706=1130.904,-110.449,-45.259,178.548,6.116,149.530
C08707=1130.899,-110.200,-45.268,178.550,6.117,149.530
C08708=1130.893,-109.950,-45.277,178.552,6.117,149.529
C08709=1130.888,-109.701,-45.285,178.554,6.117,149.529
C08710=1130.883,-109.451,-45.294,178.556,6.118,149.528
C08711=1130.877,-109.202,-45.303,178.558,6.118,149.528
C08712=1130.872,-108.951,-45.311,178.560,6.119,149.527
C08713=1130.866,-108.701,-45.321,178.562,6.120,149.527
C08714=1130.861,-108.451,-45.329,178.564,6.120,149.526
C08715=1130.856,-108.201,-45.338,178.566,6.120,149.526
C08716=1130.850,-107.952,-45.347,178.568,6.120,149.525
C08717=1130.845,-107.702,-45.356,178.570,6.121,149.525
C08718=1130.839,-107.452,-45.364,178.572,6.122,149.524
C08719=1130.834,-107.202,-45.373,178.574,6.122,149.524
C08720=1130.828,-106.953,-45.381,178.576,6.122,149.523
C08721=1130.823,-106.703,-45.390,178.577,6.122,149.523
C08722=1130.818,-106.453,-45.399,178.580,6.123,149.522
C08723=1130.813,-106.203,-45.408,178.582,6.124,149.522
C08724=1130.808,-105.953,-45.417,178.583,6.124,149.521
C08725=1130.802,-105.704,-45.426,178.586,6.125,149.521
C08726=1130.797,-105.454,-45.434,178.588,6.125,149.520
C08727=1130.792,-105.205,-45.443,178.589,6.125,149.520
C08728=1130.786,-104.955,-45.452,178.592,6.126,149.519
C08729=1130.780,-104.704,-45.461,178.593,6.126,149.519
C08730=1130.774,-104.455,-45.470,178.595,6.127,149.518
C08731=1130.769,-104.205,-45.478,178.598,6.127,149.518
C08732=1130.764,-103.955,-45.487,178.599,6.127,149.517
C08733=1130.759,-103.705,-45.496,178.601,6.128,149.517
C08734=1130.753,-103.433,-45.506,178.604,6.128,149.516
C08735=1130.748,-103.161,-45.516,178.606,6.129,149.516
C08736=1130.741,-102.889,-45.525,178.608,6.129,149.515
C08737=1130.735,-102.616,-45.535,178.610,6.130,149.515
C08738=1130.730,-102.366,-45.544,178.612,6.131,149.514
C08739=1130.724,-102.116,-45.553,178.614,6.131,149.514
C08740=1130.719,-101.866,-45.562,178.616,6.131,149.513
C08741=1130.714,-101.617,-45.571,178.618,6.132,149.513
C08742=1130.709,-101.367,-45.580,178.620,6.132,149.512
C08743=1130.703,-101.118,-45.589,178.622,6.133,149.512
C08744=1130.698,-100.868,-45.598,178.624,6.134,149.511
C08745=1130.693,-100.619,-45.607,178.626,6.134,149.511
C08746=1130.687,-100.368,-45.616,178.628,6.134,149.510
C08747=1130.682,-100.119,-45.625,178.630,6.135,149.510
C08748=1130.677,-99.869,-45.634,178.632,6.135,149.509
C08749=1130.672,-99.619,-45.643,178.634,6.136,149.509
C08750=1130.665,-99.369,-45.652,178.636,6.136,149.508
C08751=1130.660,-99.119,-45.661,178.638,6.136,149.508
C08752=1130.655,-98.870,-45.670,178.641,6.137,149.507
C08753=1130.650,-98.620,-45.679,178.642,6.137,149.507
C08754=1130.644,-98.370,-45.688,178.644,6.138,149.506
C08755=1130.639,-98.120,-45.697,178.646,6.138,149.506
C08756=1130.634,-97.871,-45.707,178.648,6.138,149.505
C08757=1130.629,-97.621,-45.716,178.650,6.139,149.505
C08758=1130.623,-97.371,-45.725,178.652,6.140,149.504
C08759=1130.617,-97.121,-45.734,178.654,6.140,149.504
C08760=1130.612,-96.872,-45.743,178.656,6.140,149.503
C08761=1130.606,-96.622,-45.751,178.658,6.141,149.503
C08762=1130.601,-96.372,-45.760,178.660,6.141,149.502
C08763=1130.596,-96.122,-45.771,178.662,6.142,149.502
C08764=1130.591,-95.872,-45.779,178.664,6.143,149.501
C08765=1130.585,-95.623,-45.788,178.666,6.143,149.501
C08766=1130.579,-95.372,-45.798,178.668,6.143,149.500
C08767=1130.574,-95.123,-45.807,178.670,6.144,149.500
C08768=1130.569,-94.873,-45.816,178.672,6.144,149.499
C08769=1130.564,-94.623,-45.825,178.674,6.145,149.499
C08770=1130.558,-94.373,-45.835,178.676,6.146,149.498
C08771=1130.553,-94.123,-45.844,178.679,6.146,149.498
C08772=1130.547,-93.874,-45.852,178.681,6.146,149.497
C08773=1130.542,-93.625,-45.862,178.683,6.147,149.497
C08774=1130.537,-93.375,-45.871,178.685,6.147,149.496
C08775=1130.532,-93.125,-45.880,178.687,6.147,149.496
C08776=1130.526,-92.875,-45.890,178.689,6.148,149.495
C08777=1130.520,-92.625,-45.899,178.691,6.149,149.495
C08778=1130.516,-92.376,-45.908,178.693,6.149,149.494
C08779=1130.510,-92.126,-45.918,178.695,6.150,149.494
C08780=1130.505,-91.876,-45.927,178.697,6.150,149.493
C08781=1130.500,-91.627,-45.936,178.699,6.150,149.493
C08782=1130.494,-91.376,-45.946,178.701,6.151,149.492
C08783=1130.489,-91.127,-45.955,178.703,6.152,149.492
C08784=1130.483,-90.877,-45.963,178.705,6.152,149.491
C08785=1130.478,-90.627,-45.974,178.707,6.152,149.491
C08786=1130.473,-90.377,-45.983,178.710,6.153,149.490
C08787=1130.468,-90.127,-45.992,178.712,6.154,149.490
C08788=1130.462,-89.878,-46.002,178.713,6.154,149.489
C08789=1130.457,-89.628,-46.011,178.715,6.154,149.489
C08790=1130.451,-89.378,-46.020,178.718,6.155,149.488
C08791=1130.446,-89.129,-46.030,178.719,6.155,149.488
C08792=1130.441,-88.879,-46.039,178.721,6.156,149.487
C08793=1130.435,-88.629,-46.049,178.724,6.156,149.487
C08794=1130.430,-88.379,-46.058,178.726,6.157,149.486
C08795=1130.424,-88.129,-46.067,178.727,6.157,149.486
C08796=1130.419,-87.880,-46.077,178.730,6.158,149.485
C08797=1130.413,-87.630,-46.086,178.732,6.159,149.485
C08798=1130.408,-87.380,-46.095,178.734,6.158,149.484
C08799=1130.403,-87.131,-46.105,178.736,6.159,149.484
C08800=1130.397,-86.881,-46.114,178.738,6.160,149.483
C08801=1130.393,-86.631,-46.124,178.741,6.161,149.483
C08802=1130.387,-86.381,-46.133,178.742,6.160,149.482
C08803=1130.382,-86.131,-46.143,178.744,6.161,149.482
C08804=1130.377,-85.881,-46.153,178.747,6.162,149.481
C08805=1130.371,-85.631,-46.162,178.749,6.163,149.481
C08806=1130.366,-85.382,-46.172,178.750,6.163,149.480
C08807=1130.361,-85.132,-46.181,178.752,6.163,149.480
C08808=1130.355,-84.882,-46.191,178.755,6.164,149.479
C08809=1130.350,-84.632,-46.200,178.757,6.164,149.479
C08810=1130.345,-84.383,-46.210,178.759,6.165,149.478
C08811=1130.339,-84.133,-46.219,178.761,6.165,149.478
C08812=1130.334,-83.884,-46.229,178.763,6.166,149.477
C08813=1130.328,-83.634,-46.238,178.765,6.166,149.477
C08814=1130.323,-83.384,-46.248,178.767,6.167,149.476
C08815=1130.318,-83.134,-46.257,178.769,6.167,149.476
C08816=1130.313,-82.884,-46.268,178.772,6.168,149.475
C08817=1130.307,-82.634,-46.277,178.773,6.168,149.475
C08818=1130.302,-82.385,-46.287,178.776,6.169,149.474
C08819=1130.297,-82.135,-46.296,178.778,6.169,149.474
C08820=1130.291,-81.885,-46.306,178.780,6.170,149.473
C08821=1130.286,-81.636,-46.316,178.782,6.170,149.473
C08822=1130.280,-81.386,-46.325,178.784,6.171,149.472
C08823=1130.275,-81.137,-46.335,178.786,6.172,149.472
C08824=1130.269,-80.886,-46.344,178.788,6.172,149.471
C08825=1130.264,-80.636,-46.355,178.790,6.172,149.471
C08826=1130.259,-80.386,-46.364,178.793,6.173,149.470
C08827=1130.254,-80.137,-46.374,178.795,6.173,149.469
C08828=1130.249,-79.888,-46.384,178.797,6.174,149.469
C08829=1130.243,-79.637,-46.393,178.799,6.174,149.468
C08830=1130.238,-79.388,-46.403,178.801,6.175,149.468
C08831=1130.232,-79.139,-46.413,178.803,6.176,149.468
C08832=1130.227,-78.889,-46.422,178.805,6.176,149.467
C08833=1130.222,-78.639,-46.432,178.807,6.176,149.467
C08834=1130.216,-78.388,-46.442,178.809,6.177,149.466
C08835=1130.211,-78.139,-46.452,178.812,6.177,149.465
C08836=1130.206,-77.890,-46.462,178.814,6.178,149.465
C08837=1130.200,-77.639,-46.471,178.816,6.179,149.464
C08838=1130.195,-77.368,-46.482,178.818,6.179,149.464
C08839=1130.189,-77.096,-46.493,178.820,6.179,149.463
C08840=1130.183,-76.825,-46.504,178.823,6.180,149.463
C08841=1130.177,-76.553,-46.514,178.825,6.181,149.462
C08842=1130.172,-76.304,-46.524,178.827,6.182,149.462
C08843=1130.166,-76.054,-46.534,178.829,6.182,149.461
C08844=1130.162,-75.804,-46.543,178.832,6.183,149.461
C08845=1130.156,-75.554,-46.554,178.833,6.183,149.460
C08846=1130.150,-75.305,-46.564,178.836,6.183,149.460
C08847=1130.145,-75.055,-46.574,178.838,6.184,149.459
C08848=1130.140,-74.805,-46.583,178.840,6.185,149.459
C08849=1130.135,-74.555,-46.594,178.842,6.186,149.458
C08850=1130.129,-74.306,-46.604,178.844,6.186,149.458
C08851=1130.124,-74.056,-46.613,178.846,6.186,149.457
C08852=1130.118,-73.806,-46.623,178.849,6.187,149.456
C08853=1130.113,-73.557,-46.633,178.851,6.188,149.456
C08854=1130.108,-73.306,-46.644,178.853,6.188,149.455
C08855=1130.103,-73.057,-46.653,178.855,6.188,149.455
C08856=1130.097,-72.808,-46.663,178.857,6.189,149.455
C08857=1130.091,-72.557,-46.673,178.859,6.190,149.454
C08858=1130.087,-72.307,-46.683,178.862,6.190,149.453
C08859=1130.081,-72.058,-46.693,178.864,6.191,149.453
C08860=1130.076,-71.808,-46.703,178.865,6.191,149.452
C08861=1130.070,-71.559,-46.714,178.868,6.192,149.452
C08862=1130.065,-71.309,-46.724,178.870,6.192,149.451
C08863=1130.060,-71.059,-46.733,178.872,6.193,149.451
C08864=1130.054,-70.809,-46.743,178.875,6.193,149.450
C08865=1130.049,-70.560,-46.753,178.876,6.193,149.450
C08866=1130.044,-70.309,-46.764,178.878,6.194,149.449
C08867=1130.039,-70.060,-46.774,178.881,6.195,149.449
C08868=1130.033,-69.811,-46.784,178.883,6.196,149.448
C08869=1130.028,-69.561,-46.794,178.885,6.196,149.448
C08870=1130.023,-69.311,-46.805,178.887,6.196,149.447
C08871=1130.017,-69.061,-46.815,178.889,6.197,149.447
C08872=1130.012,-68.811,-46.824,178.892,6.198,149.446
C08873=1130.007,-68.561,-46.834,178.894,6.198,149.446
C08874=1130.001,-68.312,-46.845,178.896,6.199,149.445
C08875=1129.996,-68.062,-46.855,178.898,6.200,149.445
C08876=1129.990,-67.813,-46.865,178.900,6.200,149.444
C08877=1129.985,-67.562,-46.876,178.902,6.200,149.444
C08878=1129.980,-67.313,-46.885,178.905,6.201,149.443
C08879=1129.975,-67.064,-46.895,178.907,6.202,149.443
C08880=1129.970,-66.813,-46.906,178.909,6.202,149.442
C08881=1129.964,-66.564,-46.916,178.911,6.203,149.442
C08882=1129.959,-66.314,-46.926,178.913,6.203,149.441
C08883=1129.954,-66.064,-46.937,178.915,6.204,149.440
C08884=1129.948,-65.814,-46.947,178.918,6.204,149.440
C08885=1129.943,-65.565,-46.957,178.920,6.205,149.439
C08886=1129.938,-65.315,-46.967,178.922,6.206,149.439
C08887=1129.933,-65.065,-46.978,178.924,6.207,149.438
C08888=1129.927,-64.816,-46.988,178.927,6.207,149.438
C08889=1129.922,-64.566,-46.998,178.928,6.207,149.437
C08890=1129.916,-64.316,-47.009,178.931,6.208,149.437
C08891=1129.911,-64.067,-47.019,178.933,6.209,149.436
C08892=1129.906,-63.816,-47.029,178.935,6.209,149.436
C08893=1129.900,-63.567,-47.040,178.937,6.210,149.435
C08894=1129.895,-63.317,-47.051,178.940,6.210,149.435
C08895=1129.890,-63.068,-47.061,178.941,6.210,149.434
C08896=1129.885,-62.818,-47.071,178.944,6.211,149.434
C08897=1129.880,-62.568,-47.081,178.946,6.212,149.433
C08898=1129.874,-62.319,-47.091,178.948,6.213,149.433
C08899=1129.869,-62.069,-47.102,178.951,6.213,149.432
C08900=1129.864,-61.819,-47.112,178.953,6.214,149.432
C08901=1129.858,-61.569,-47.122,178.955,6.215,149.431
C08902=1129.853,-61.319,-47.133,178.957,6.215,149.431
C08903=1129.848,-61.070,-47.144,178.959,6.215,149.430
C08904=1129.842,-60.821,-47.154,178.962,6.216,149.429
C08905=1129.837,-60.570,-47.165,178.964,6.216,149.429
C08906=1129.832,-60.321,-47.175,178.966,6.217,149.428
C08907=1129.827,-60.071,-47.185,178.968,6.218,149.428
C08908=1129.821,-59.821,-47.196,178.970,6.219,149.427
C08909=1129.816,-59.571,-47.207,178.973,6.219,149.427
C08910=1129.811,-59.322,-47.217,178.975,6.220,149.426
C08911=1129.805,-59.072,-47.227,178.977,6.220,149.426
C08912=1129.800,-58.822,-47.238,178.979,6.221,149.425
C08913=1129.795,-58.572,-47.248,178.981,6.221,149.425
C08914=1129.790,-58.323,-47.259,178.983,6.222,149.424
C08915=1129.784,-58.073,-47.270,178.986,6.222,149.424
C08916=1129.779,-57.823,-47.280,178.988,6.223,149.423
C08917=1129.774,-57.574,-47.290,178.990,6.224,149.423
C08918=1129.769,-57.324,-47.302,178.993,6.225,149.422
C08919=1129.764,-57.074,-47.312,178.995,6.226,149.422
C08920=1129.758,-56.825,-47.322,178.997,6.225,149.421
C08921=1129.753,-56.575,-47.333,178.999,6.226,149.421
C08922=1129.748,-56.326,-47.344,179.001,6.227,149.420
C08923=1129.742,-56.075,-47.355,179.003,6.227,149.420
C08924=1129.736,-55.826,-47.365,179.006,6.228,149.419
C08925=1129.732,-55.576,-47.376,179.008,6.229,149.418
C08926=1129.726,-55.326,-47.387,179.010,6.229,149.418
C08927=1129.721,-55.076,-47.397,179.013,6.230,149.417
C08928=1129.716,-54.827,-47.408,179.015,6.231,149.417
C08929=1129.711,-54.577,-47.419,179.018,6.231,149.416
C08930=1129.705,-54.327,-47.429,179.019,6.231,149.416
C08931=1129.700,-54.078,-47.440,179.021,6.232,149.415
C08932=1129.695,-53.828,-47.450,179.023,6.233,149.415
C08933=1129.689,-53.578,-47.461,179.026,6.234,149.414
C08934=1129.684,-53.329,-47.472,179.028,6.234,149.414
C08935=1129.679,-53.079,-47.483,179.031,6.235,149.413
C08936=1129.673,-52.830,-47.494,179.033,6.235,149.413
C08937=1129.669,-52.579,-47.504,179.035,6.236,149.412
C08938=1129.663,-52.330,-47.515,179.037,6.237,149.412
C08939=1129.658,-52.080,-47.526,179.040,6.237,149.411
C08940=1129.652,-51.830,-47.537,179.042,6.238,149.411
C08941=1129.647,-51.581,-47.548,179.044,6.239,149.410
C08942=1129.641,-51.309,-47.560,179.046,6.240,149.410
C08943=1129.636,-51.039,-47.571,179.049,6.240,149.409
C08944=1129.630,-50.768,-47.583,179.051,6.241,149.408
C08945=1129.625,-50.497,-47.595,179.054,6.241,149.408
C08946=1129.619,-50.248,-47.606,179.056,6.242,149.407
C08947=1129.614,-49.998,-47.617,179.058,6.243,149.407
C08948=1129.609,-49.748,-47.627,179.060,6.243,149.406
C08949=1129.603,-49.499,-47.639,179.063,6.244,149.406
C08950=1129.598,-49.249,-47.649,179.065,6.245,149.405
C08951=1129.593,-48.999,-47.660,179.068,6.245,149.405
C08952=1129.588,-48.749,-47.671,179.069,6.245,149.404
C08953=1129.582,-48.500,-47.683,179.071,6.246,149.404
C08954=1129.577,-48.250,-47.693,179.074,6.247,149.403
C08955=1129.572,-48.001,-47.704,179.076,6.247,149.402
C08956=1129.567,-47.750,-47.715,179.078,6.248,149.402
C08957=1129.561,-47.501,-47.727,179.081,6.249,149.401
C08958=1129.556,-47.251,-47.737,179.083,6.249,149.401
C08959=1129.551,-47.001,-47.748,179.085,6.250,149.400
C08960=1129.545,-46.751,-47.759,179.088,6.251,149.400
C08961=1129.540,-46.502,-47.770,179.090,6.252,149.399
C08962=1129.535,-46.252,-47.781,179.092,6.252,149.399
C08963=1129.530,-46.003,-47.792,179.095,6.253,149.398
C08964=1129.524,-45.753,-47.804,179.097,6.253,149.398
C08965=1129.519,-45.503,-47.814,179.099,6.254,149.397
C08966=1129.514,-45.254,-47.825,179.101,6.255,149.397
C08967=1129.508,-45.004,-47.837,179.104,6.255,149.396
C08968=1129.503,-44.754,-47.847,179.106,6.256,149.396
C08969=1129.498,-44.504,-47.858,179.108,6.257,149.395
C08970=1129.493,-44.255,-47.870,179.110,6.258,149.395
C08971=1129.487,-44.005,-47.880,179.113,6.258,149.394
C08972=1129.482,-43.755,-47.892,179.115,6.259,149.393
C08973=1129.477,-43.505,-47.904,179.117,6.260,149.393
C08974=1129.471,-43.256,-47.914,179.120,6.260,149.392
C08975=1129.467,-43.006,-47.925,179.122,6.261,149.392
C08976=1129.461,-42.756,-47.937,179.125,6.262,149.391
C08977=1129.456,-42.507,-47.947,179.127,6.262,149.391
C08978=1129.450,-42.257,-47.959,179.129,6.263,149.390
C08979=1129.446,-42.007,-47.970,179.132,6.263,149.390
C08980=1129.440,-41.758,-47.981,179.134,6.264,149.389
C08981=1129.435,-41.508,-47.993,179.136,6.265,149.389
C08982=1129.430,-41.258,-48.004,179.138,6.266,149.388
C08983=1129.424,-41.009,-48.015,179.140,6.267,149.388
C08984=1129.419,-40.759,-48.027,179.143,6.267,149.387
C08985=1129.414,-40.509,-48.037,179.145,6.268,149.387
C08986=1129.409,-40.259,-48.049,179.147,6.268,149.386
C08987=1129.403,-40.010,-48.060,179.149,6.268,149.386
C08988=1129.398,-39.760,-48.072,179.152,6.269,149.385
C08989=1129.393,-39.511,-48.083,179.154,6.270,149.384
C08990=1129.387,-39.261,-48.094,179.157,6.271,149.384
C08991=1129.382,-39.011,-48.105,179.159,6.272,149.383
C08992=1129.377,-38.761,-48.117,179.161,6.272,149.383
C08993=1129.372,-38.512,-48.128,179.164,6.273,149.382
C08994=1129.366,-38.262,-48.140,179.166,6.274,149.382
C08995=1129.361,-38.013,-48.151,179.168,6.275,149.381
C08996=1129.356,-37.762,-48.162,179.171,6.275,149.381
C08997=1129.350,-37.513,-48.173,179.173,6.276,149.380
C08998=1129.345,-37.263,-48.185,179.175,6.277,149.380
C08999=1129.340,-37.014,-48.197,179.177,6.277,149.379
C09000=1129.335,-36.764,-48.208,179.180,6.278,149.378
C09001=1129.330,-36.515,-48.219,179.182,6.279,149.378
C09002=1129.324,-36.265,-48.231,179.184,6.279,149.378
C09003=1129.319,-36.015,-48.243,179.186,6.280,149.377
C09004=1129.314,-35.765,-48.254,179.189,6.281,149.376
C09005=1129.309,-35.515,-48.265,179.191,6.281,149.376
C09006=1129.303,-35.266,-48.276,179.194,6.282,149.375
C09007=1129.298,-35.016,-48.288,179.196,6.283,149.375
C09008=1129.293,-34.766,-48.300,179.198,6.283,149.374
C09009=1129.288,-34.517,-48.311,179.201,6.284,149.374
C09010=1129.283,-34.267,-48.323,179.203,6.285,149.373
C09011=1129.277,-34.017,-48.334,179.205,6.286,149.373
C09012=1129.272,-33.768,-48.346,179.208,6.286,149.372
C09013=1129.267,-33.518,-48.358,179.210,6.287,149.372
C09014=1129.262,-33.268,-48.369,179.212,6.288,149.371
C09015=1129.256,-33.018,-48.381,179.215,6.288,149.370
C09016=1129.251,-32.769,-48.392,179.217,6.289,149.370
C09017=1129.246,-32.519,-48.404,179.219,6.289,149.370
C09018=1129.240,-32.270,-48.415,179.221,6.290,149.369
C09019=1129.236,-32.020,-48.427,179.224,6.291,149.368
C09020=1129.230,-31.770,-48.439,179.226,6.291,149.368
C09021=1129.225,-31.520,-48.450,179.228,6.292,149.367
C09022=1129.219,-31.271,-48.461,179.230,6.293,149.367
C09023=1129.214,-31.022,-48.474,179.233,6.293,149.366
C09024=1129.210,-30.772,-48.485,179.236,6.295,149.366
C09025=1129.204,-30.522,-48.497,179.238,6.296,149.365
C09026=1129.199,-30.272,-48.509,179.240,6.296,149.365
C09027=1129.194,-30.023,-48.520,179.243,6.297,149.364
C09028=1129.189,-29.773,-48.532,179.245,6.298,149.364
C09029=1129.183,-29.523,-48.544,179.247,6.298,149.363
C09030=1129.178,-29.274,-48.555,179.249,6.299,149.363
C09031=1129.172,-29.024,-48.567,179.252,6.300,149.362
C09032=1129.167,-28.775,-48.580,179.254,6.300,149.361
C09033=1129.163,-28.525,-48.591,179.257,6.301,149.361
C09034=1129.157,-28.275,-48.603,179.259,6.302,149.361
C09035=1129.152,-28.025,-48.615,179.261,6.302,149.360
C09036=1129.146,-27.775,-48.626,179.264,6.303,149.359
C09037=1129.142,-27.526,-48.638,179.266,6.304,149.359
C09038=1129.136,-27.277,-48.650,179.269,6.305,149.358
C09039=1129.131,-27.027,-48.662,179.271,6.306,149.358
C09040=1129.126,-26.777,-48.673,179.273,6.307,149.357
C09041=1129.120,-26.527,-48.685,179.276,6.307,149.357
C09042=1129.115,-26.277,-48.697,179.278,6.308,149.356
C09043=1129.110,-26.028,-48.710,179.280,6.309,149.356
C09044=1129.105,-25.779,-48.721,179.283,6.309,149.355
C09045=1129.100,-25.529,-48.733,179.285,6.310,149.355
C09046=1129.094,-25.258,-48.746,179.287,6.311,149.354
C09047=1129.089,-24.989,-48.758,179.290,6.312,149.353
C09048=1129.082,-24.718,-48.772,179.293,6.313,149.353
C09049=1129.077,-24.448,-48.785,179.295,6.313,149.352
C09050=1129.072,-24.199,-48.796,179.298,6.314,149.352
C09051=1129.067,-23.949,-48.808,179.300,6.314,149.351
C09052=1129.061,-23.699,-48.820,179.303,6.316,149.351
C09053=1129.056,-23.449,-48.832,179.305,6.317,149.350
C09054=1129.051,-23.200,-48.845,179.308,6.317,149.349
C09055=1129.045,-22.950,-48.857,179.310,6.318,149.349
C09056=1129.041,-22.701,-48.868,179.312,6.319,149.349
C09057=1129.036,-22.451,-48.880,179.314,6.320,149.348
C09058=1129.030,-22.201,-48.892,179.317,6.320,149.347
C09059=1129.025,-21.951,-48.904,179.319,6.321,149.347
C09060=1129.020,-21.702,-48.917,179.321,6.322,149.346
C09061=1129.014,-21.452,-48.929,179.324,6.323,149.346
C09062=1129.009,-21.203,-48.941,179.327,6.324,149.345
C09063=1129.004,-20.953,-48.953,179.329,6.324,149.345
C09064=1128.999,-20.703,-48.965,179.331,6.325,149.344
C09065=1128.994,-20.454,-48.977,179.334,6.325,149.344
C09066=1128.988,-20.204,-48.989,179.336,6.326,149.343
C09067=1128.983,-19.955,-49.002,179.338,6.327,149.343
C09068=1128.978,-19.705,-49.013,179.341,6.327,149.342
C09069=1128.973,-19.455,-49.026,179.343,6.329,149.342
C09070=1128.967,-19.206,-49.038,179.346,6.330,149.341
C09071=1128.962,-18.956,-49.050,179.348,6.331,149.341
C09072=1128.957,-18.706,-49.062,179.350,6.331,149.340
C09073=1128.951,-18.456,-49.074,179.353,6.332,149.339
C09074=1128.929,-17.334,-49.132,179.540,6.000,149.212
C09075=1128.924,-17.085,-49.144,179.541,6.004,149.212
C09076=1128.918,-16.835,-49.156,179.542,6.009,149.213
C09077=1128.914,-16.586,-49.168,179.542,6.013,149.214
C09078=1128.908,-16.336,-49.180,179.543,6.019,149.215
C09079=1128.903,-16.087,-49.193,179.544,6.023,149.216
C09080=1128.898,-15.837,-49.204,179.545,6.028,149.216
C09081=1128.893,-15.588,-49.217,179.545,6.033,149.217
C09082=1128.887,-15.338,-49.229,179.546,6.037,149.218
C09083=1128.882,-15.088,-49.242,179.547,6.042,149.219
C09084=1128.877,-14.838,-49.253,179.548,6.047,149.220
C09085=1128.871,-14.589,-49.266,179.549,6.052,149.220
C09086=1128.867,-14.339,-49.279,179.549,6.056,149.221
C09087=1128.862,-14.089,-49.291,179.550,6.061,149.222
C09088=1128.856,-13.840,-49.303,179.551,6.066,149.223
C09089=1128.851,-13.590,-49.315,179.551,6.070,149.224
C09090=1128.846,-13.341,-49.328,179.552,6.075,149.224
C09091=1128.841,-13.091,-49.341,179.553,6.079,149.225
C09092=1128.835,-12.841,-49.352,179.553,6.084,149.226
C09093=1128.830,-12.592,-49.365,179.555,6.089,149.227
C09094=1128.825,-12.342,-49.379,179.555,6.094,149.228
C09095=1128.819,-12.092,-49.390,179.556,6.099,149.229
C09096=1128.814,-11.842,-49.403,179.557,6.103,149.229
C09097=1128.809,-11.593,-49.416,179.557,6.108,149.230
C09098=1128.804,-11.343,-49.428,179.558,6.112,149.231
C09099=1128.799,-11.094,-49.440,179.559,6.117,149.232
C09100=1128.794,-10.845,-49.453,179.559,6.122,149.233
C09101=1128.789,-10.595,-49.466,179.560,6.126,149.233
C09102=1128.784,-10.345,-49.478,179.561,6.131,149.234
C09103=1128.778,-10.095,-49.490,179.561,6.135,149.235
C09104=1128.773,-9.846,-49.503,179.562,6.140,149.236
C09105=1128.767,-9.596,-49.516,179.563,6.144,149.237
C09106=1128.763,-9.346,-49.528,179.563,6.149,149.237
C09107=1128.758,-9.096,-49.541,179.564,6.153,149.238
C09108=1128.752,-8.847,-49.553,179.565,6.158,149.239
C09109=1128.747,-8.598,-49.566,179.566,6.163,149.240
C09110=1128.742,-8.348,-49.579,179.566,6.167,149.241
C09111=1128.737,-8.098,-49.592,179.567,6.172,149.241
C09112=1128.731,-7.848,-49.604,179.568,6.176,149.242
C09113=1128.726,-7.599,-49.617,179.568,6.181,149.243
C09114=1128.721,-7.350,-49.629,179.569,6.186,149.244
C09115=1128.716,-7.118,-49.641,179.570,6.190,149.245
C09116=1128.712,-6.887,-49.653,179.570,6.194,149.245
C09117=1128.707,-6.658,-49.665,179.571,6.198,149.246
C09118=1128.702,-6.426,-49.677,179.572,6.203,149.247
C09119=1128.698,-6.195,-49.689,179.572,6.207,149.248
C09120=1128.693,-5.965,-49.700,179.573,6.211,149.248
C09121=1128.688,-5.734,-49.712,179.573,6.215,149.249
C09122=1128.684,-5.504,-49.724,179.574,6.219,149.250
C09123=1128.678,-5.254,-49.737,179.575,6.224,149.250
C09124=1128.673,-5.005,-49.750,179.575,6.228,149.251
C09125=1128.667,-4.755,-49.763,179.576,6.233,149.252
C09126=1128.663,-4.505,-49.775,179.576,6.238,149.253
C09127=1128.657,-4.256,-49.789,179.577,6.242,149.254
C09128=1128.652,-4.006,-49.801,179.578,6.247,149.255
